C05385=1038.334,449.615,-148.521,176.484,47.158,159.856
C05386=1038.308,449.370,-148.478,176.465,47.152,159.852
C05387=1038.284,449.126,-148.433,176.446,47.146,159.848
C05388=1038.259,448.881,-148.389,176.428,47.139,159.843
C05389=1038.236,448.635,-148.344,176.409,47.132,159.839
C05390=1038.213,448.391,-148.298,176.390,47.125,159.834
C05391=1038.190,448.146,-148.252,176.372,47.118,159.830
C05392=1038.168,447.901,-148.206,176.353,47.112,159.825
C05393=1038.146,447.657,-148.159,176.335,47.105,159.821
C05394=1038.125,447.413,-148.112,176.318,47.097,159.816
C05395=1038.105,447.168,-148.064,176.299,47.090,159.812
C05396=1038.085,446.924,-148.016,176.281,47.083,159.807
C05397=1038.065,446.680,-147.967,176.264,47.076,159.803
C05398=1038.047,446.435,-147.918,176.245,47.068,159.798
C05399=1038.029,446.191,-147.869,176.228,47.060,159.794
C05400=1038.012,445.948,-147.819,176.211,47.053,159.789
C05401=1037.994,445.705,-147.768,176.192,47.045,159.785
C05402=1037.978,445.460,-147.718,176.174,47.037,159.780
C05403=1037.962,445.217,-147.666,176.157,47.029,159.776
C05404=1037.946,444.973,-147.614,176.141,47.021,159.771
C05405=1037.932,444.730,-147.563,176.123,47.013,159.766
C05406=1037.917,444.485,-147.509,176.105,47.005,159.762
C05407=1037.904,444.241,-147.456,176.089,46.996,159.757
C05408=1037.890,443.996,-147.402,176.071,46.988,159.752
C05409=1037.877,443.752,-147.349,176.054,46.979,159.747
C05410=1037.863,443.508,-147.296,176.038,46.971,159.743
C05411=1037.849,443.264,-147.243,176.020,46.963,159.738
C05412=1037.836,443.020,-147.189,176.004,46.955,159.734
C05413=1037.823,442.776,-147.136,175.987,46.946,159.729
C05414=1037.810,442.532,-147.082,175.971,46.938,159.725
C05415=1037.797,442.288,-147.029,175.954,46.930,159.720
C05416=1037.783,442.044,-146.977,175.937,46.922,159.716
C05417=1037.770,441.800,-146.924,175.920,46.914,159.711
C05418=1037.757,441.556,-146.871,175.904,46.905,159.707
C05419=1037.744,441.312,-146.818,175.888,46.897,159.702
C05420=1037.732,441.068,-146.766,175.871,46.889,159.698
C05421=1037.718,440.824,-146.712,175.855,46.881,159.693
C05422=1037.705,440.581,-146.660,175.839,46.873,159.689
C05423=1037.692,440.336,-146.607,175.824,46.865,159.685
C05424=1037.679,440.091,-146.555,175.807,46.857,159.680
C05425=1037.667,439.848,-146.502,175.791,46.849,159.676
C05426=1037.653,439.604,-146.450,175.775,46.841,159.671
C05427=1037.640,439.359,-146.398,175.759,46.833,159.667
C05428=1037.628,439.115,-146.346,175.744,46.825,159.663
C05429=1037.615,438.871,-146.293,175.728,46.817,159.659
C05430=1037.602,438.627,-146.241,175.712,46.809,159.654
C05431=1037.590,438.383,-146.189,175.697,46.802,159.650
C05432=1037.577,438.138,-146.137,175.681,46.794,159.646
C05433=1037.564,437.895,-146.085,175.665,46.786,159.642
C05434=1037.552,437.653,-146.034,175.650,46.778,159.638
C05435=1037.539,437.412,-145.983,175.635,46.771,159.634
C05436=1037.527,437.170,-145.931,175.619,46.763,159.629
C05437=1037.514,436.929,-145.880,175.605,46.755,159.625
C05438=1037.502,436.688,-145.829,175.590,46.748,159.621
C05439=1037.489,436.446,-145.778,175.574,46.740,159.617
C05440=1037.477,436.205,-145.726,175.560,46.733,159.613
C05441=1037.465,435.963,-145.676,175.545,46.725,159.609
C05442=1037.453,435.719,-145.624,175.530,46.718,159.605
C05443=1037.439,435.474,-145.573,175.514,46.710,159.601
C05444=1037.428,435.230,-145.521,175.500,46.703,159.597
C05445=1037.416,434.985,-145.470,175.485,46.696,159.593
C05446=1037.403,434.741,-145.419,175.470,46.688,159.589
C05447=1037.391,434.497,-145.368,175.455,46.681,159.585
C05448=1037.379,434.252,-145.317,175.440,46.673,159.581
C05449=1037.365,434.007,-145.266,175.426,46.666,159.577
C05450=1037.353,433.763,-145.214,175.411,46.658,159.574
C05451=1037.341,433.519,-145.164,175.397,46.651,159.570
C05452=1037.329,433.274,-145.113,175.382,46.644,159.566
C05453=1037.317,433.029,-145.062,175.368,46.637,159.562
C05454=1037.304,432.785,-145.011,175.354,46.629,159.558
C05455=1037.292,432.540,-144.961,175.339,46.622,159.554
C05456=1037.280,432.297,-144.910,175.325,46.615,159.551
C05457=1037.268,432.052,-144.860,175.310,46.607,159.547
C05458=1037.256,431.807,-144.809,175.296,46.601,159.543
C05459=1037.244,431.562,-144.758,175.283,46.593,159.539
C05460=1037.232,431.317,-144.708,175.268,46.586,159.535
C05461=1037.220,431.072,-144.658,175.254,46.579,159.532
C05462=1037.208,430.829,-144.607,175.240,46.572,159.528
C05463=1037.196,430.584,-144.557,175.226,46.565,159.524
C05464=1037.184,430.339,-144.506,175.213,46.558,159.521
C05465=1037.173,430.095,-144.456,175.199,46.551,159.517
C05466=1037.161,429.850,-144.406,175.184,46.544,159.513
C05467=1037.149,429.606,-144.356,175.171,46.537,159.510
C05468=1037.138,429.360,-144.306,175.157,46.530,159.506
C05469=1037.125,429.116,-144.256,175.144,46.523,159.502
C05470=1037.114,428.871,-144.207,175.130,46.516,159.499
C05471=1037.103,428.626,-144.156,175.117,46.509,159.495
C05472=1037.091,428.382,-144.106,175.103,46.503,159.492
C05473=1037.080,428.137,-144.056,175.090,46.495,159.488
C05474=1037.068,427.892,-144.006,175.076,46.489,159.485
C05475=1037.056,427.648,-143.957,175.063,46.482,159.481
C05476=1037.044,427.402,-143.907,175.049,46.475,159.478
C05477=1037.033,427.157,-143.858,175.036,46.468,159.474
C05478=1037.022,426.913,-143.808,175.023,46.462,159.471
C05479=1037.010,426.668,-143.759,175.010,46.455,159.467
C05480=1036.998,426.423,-143.710,174.997,46.448,159.464
C05481=1036.987,426.178,-143.661,174.984,46.442,159.460
C05482=1036.975,425.933,-143.611,174.970,46.435,159.457
C05483=1036.963,425.689,-143.561,174.957,46.428,159.453
C05484=1036.952,425.444,-143.512,174.944,46.422,159.450
C05485=1036.941,425.199,-143.463,174.932,46.415,159.447
C05486=1036.930,424.953,-143.415,174.919,46.409,159.443
C05487=1036.918,424.709,-143.366,174.905,46.402,159.440
C05488=1036.907,424.464,-143.316,174.892,46.395,159.436
C05489=1036.896,424.219,-143.267,174.880,46.389,159.433
C05490=1036.884,423.974,-143.218,174.867,46.383,159.430
C05491=1036.873,423.730,-143.169,174.855,46.376,159.427
C05492=1036.861,423.484,-143.121,174.842,46.370,159.423
C05493=1036.850,423.239,-143.072,174.830,46.364,159.420
C05494=1036.839,423.000,-143.024,174.817,46.357,159.417
C05495=1036.828,422.760,-142.977,174.805,46.351,159.414
C05496=1036.817,422.521,-142.930,174.793,46.345,159.411
C05497=1036.806,422.281,-142.882,174.781,46.339,159.408
C05498=1036.795,422.041,-142.835,174.769,46.333,159.404
C05499=1036.784,421.802,-142.788,174.756,46.326,159.401
C05500=1036.774,421.562,-142.741,174.745,46.320,159.398
C05501=1036.763,421.322,-142.693,174.732,46.314,159.395
C05502=1036.752,421.077,-142.645,174.720,46.308,159.392
C05503=1036.740,420.833,-142.598,174.708,46.302,159.389
C05504=1036.729,420.588,-142.549,174.696,46.296,159.386
C05505=1036.718,420.343,-142.500,174.684,46.290,159.382
C05506=1036.708,420.097,-142.453,174.672,46.283,159.379
C05507=1036.697,419.852,-142.405,174.659,46.278,159.376
C05508=1036.685,419.607,-142.356,174.648,46.271,159.373
C05509=1036.675,419.362,-142.309,174.636,46.265,159.370
C05510=1036.664,419.117,-142.260,174.623,46.259,159.367
C05511=1036.653,418.871,-142.212,174.612,46.253,159.364
C05512=1036.642,418.626,-142.165,174.600,46.247,159.361
C05513=1036.631,418.381,-142.117,174.589,46.241,159.358
C05514=1036.620,418.136,-142.069,174.576,46.235,159.355
C05515=1036.610,417.891,-142.022,174.565,46.229,159.352
C05516=1036.599,417.646,-141.974,174.553,46.223,159.349
C05517=1036.589,417.400,-141.926,174.541,46.217,159.346
C05518=1036.577,417.155,-141.879,174.530,46.211,159.343
C05519=1036.567,416.910,-141.831,174.518,46.205,159.340
C05520=1036.556,416.664,-141.784,174.507,46.200,159.337
C05521=1036.545,416.419,-141.737,174.496,46.194,159.334
C05522=1036.535,416.174,-141.689,174.484,46.188,159.331
C05523=1036.523,415.929,-141.642,174.473,46.182,159.328
C05524=1036.513,415.683,-141.595,174.461,46.177,159.325
C05525=1036.503,415.438,-141.548,174.450,46.171,159.322
C05526=1036.491,415.192,-141.501,174.439,46.165,159.320
C05527=1036.481,414.947,-141.454,174.427,46.160,159.317
C05528=1036.470,414.702,-141.407,174.416,46.154,159.314
C05529=1036.460,414.457,-141.360,174.405,46.148,159.311
C05530=1036.450,414.212,-141.313,174.393,46.142,159.308
C05531=1036.438,413.965,-141.266,174.382,46.137,159.305
C05532=1036.428,413.720,-141.219,174.371,46.131,159.303
C05533=1036.417,413.475,-141.173,174.360,46.126,159.300
C05534=1036.407,413.230,-141.125,174.349,46.120,159.297
C05535=1036.397,412.984,-141.079,174.337,46.114,159.294
C05536=1036.386,412.739,-141.032,174.327,46.109,159.291
C05537=1036.376,412.494,-140.985,174.316,46.103,159.289
C05538=1036.365,412.248,-140.939,174.305,46.098,159.286
C05539=1036.355,412.003,-140.892,174.294,46.093,159.283
C05540=1036.345,411.757,-140.845,174.284,46.087,159.281
C05541=1036.334,411.512,-140.799,174.272,46.082,159.278
C05542=1036.325,411.266,-140.752,174.261,46.076,159.275
C05543=1036.314,411.020,-140.706,174.250,46.070,159.272
C05544=1036.303,410.775,-140.660,174.240,46.065,159.270
C05545=1036.293,410.529,-140.614,174.229,46.060,159.267
C05546=1036.283,410.285,-140.568,174.218,46.055,159.264
C05547=1036.272,410.039,-140.522,174.208,46.049,159.262
C05548=1036.262,409.793,-140.476,174.197,46.044,159.259
C05549=1036.252,409.547,-140.429,174.186,46.039,159.256
C05550=1036.241,409.302,-140.383,174.176,46.034,159.254
C05551=1036.231,409.057,-140.338,174.165,46.028,159.251
C05552=1036.221,408.811,-140.293,174.155,46.023,159.249
C05553=1036.211,408.565,-140.246,174.145,46.018,159.246
C05554=1036.201,408.330,-140.202,174.135,46.013,159.244
C05555=1036.192,408.095,-140.159,174.124,46.008,159.241
C05556=1036.181,407.860,-140.114,174.115,46.003,159.239
C05557=1036.172,407.624,-140.071,174.105,45.998,159.236
C05558=1036.162,407.390,-140.028,174.095,45.993,159.234
C05559=1036.152,407.155,-139.984,174.085,45.988,159.231
C05560=1036.144,406.919,-139.940,174.076,45.983,159.229
C05561=1036.133,406.683,-139.896,174.065,45.979,159.227
C05562=1036.123,406.439,-139.850,174.056,45.973,159.224
C05563=1036.113,406.192,-139.805,174.045,45.968,159.222
C05564=1036.103,405.947,-139.760,174.035,45.963,159.219
C05565=1036.093,405.701,-139.714,174.025,45.959,159.217
C05566=1036.084,405.455,-139.669,174.015,45.953,159.214
C05567=1036.074,405.211,-139.623,174.005,45.948,159.212
C05568=1036.063,404.964,-139.578,173.995,45.944,159.209
C05569=1036.054,404.719,-139.533,173.985,45.938,159.207
C05570=1036.044,404.474,-139.487,173.975,45.933,159.204
C05571=1036.034,404.227,-139.442,173.964,45.929,159.202
C05572=1036.024,403.982,-139.397,173.955,45.923,159.199
C05573=1036.015,403.736,-139.352,173.945,45.919,159.197
C05574=1036.005,403.490,-139.307,173.936,45.914,159.195
C05575=1035.995,403.244,-139.262,173.925,45.909,159.192
C05576=1035.986,402.999,-139.217,173.916,45.904,159.190
C05577=1035.976,402.753,-139.172,173.906,45.899,159.188
C05578=1035.966,402.508,-139.127,173.896,45.894,159.185
C05579=1035.956,402.262,-139.082,173.886,45.889,159.183
C05580=1035.946,402.016,-139.037,173.877,45.885,159.181
C05581=1035.936,401.771,-138.993,173.867,45.880,159.178
C05582=1035.927,401.525,-138.948,173.858,45.875,159.176
C05583=1035.917,401.279,-138.904,173.848,45.871,159.174
C05584=1035.908,401.033,-138.859,173.838,45.866,159.171
C05585=1035.898,400.788,-138.814,173.828,45.861,159.169
C05586=1035.889,400.542,-138.770,173.819,45.856,159.167
C05587=1035.879,400.296,-138.725,173.809,45.852,159.164
C05588=1035.869,400.050,-138.681,173.800,45.848,159.162
C05589=1035.860,399.805,-138.636,173.791,45.843,159.160
C05590=1035.850,399.558,-138.592,173.781,45.838,159.158
C05591=1035.841,399.313,-138.547,173.772,45.833,159.155
C05592=1035.830,399.067,-138.504,173.763,45.829,159.153
C05593=1035.821,398.822,-138.459,173.753,45.825,159.151
C05594=1035.811,398.575,-138.415,173.743,45.820,159.149
C05595=1035.802,398.329,-138.371,173.735,45.815,159.146
C05596=1035.792,398.083,-138.327,173.724,45.811,159.144
C05597=1035.783,397.838,-138.283,173.716,45.807,159.142
C05598=1035.773,397.593,-138.239,173.707,45.802,159.140
C05599=1035.764,397.346,-138.194,173.697,45.798,159.138
C05600=1035.754,397.100,-138.150,173.688,45.793,159.135
C05601=1035.744,396.854,-138.107,173.679,45.789,159.133
C05602=1035.735,396.609,-138.063,173.670,45.784,159.131
C05603=1035.726,396.363,-138.019,173.661,45.780,159.129
C05604=1035.717,396.117,-137.975,173.651,45.776,159.127
C05605=1035.706,395.871,-137.931,173.642,45.772,159.125
C05606=1035.698,395.626,-137.888,173.633,45.767,159.122
C05607=1035.688,395.379,-137.843,173.624,45.762,159.120
C05608=1035.679,395.133,-137.800,173.615,45.758,159.118
C05609=1035.670,394.888,-137.757,173.606,45.754,159.116
C05610=1035.660,394.641,-137.713,173.597,45.750,159.114
C05611=1035.651,394.396,-137.669,173.588,45.745,159.112
C05612=1035.642,394.150,-137.626,173.579,45.741,159.110
C05613=1035.632,393.903,-137.582,173.570,45.737,159.108
C05614=1035.623,393.678,-137.543,173.563,45.733,159.106
C05615=1035.616,393.453,-137.503,173.554,45.729,159.104
C05616=1035.607,393.228,-137.464,173.545,45.725,159.102
C05617=1035.598,393.003,-137.424,173.538,45.722,159.100
C05618=1035.590,392.778,-137.384,173.530,45.718,159.098
C05619=1035.581,392.553,-137.345,173.522,45.714,159.097
C05620=1035.573,392.328,-137.305,173.514,45.710,159.095
C05621=1035.565,392.103,-137.265,173.506,45.706,159.093
C05622=1035.555,391.857,-137.223,173.497,45.702,159.091
C05623=1035.546,391.611,-137.179,173.489,45.698,159.089
C05624=1035.537,391.366,-137.136,173.480,45.694,159.087
C05625=1035.528,391.120,-137.093,173.471,45.690,159.085
C05626=1035.519,390.873,-137.050,173.462,45.686,159.083
C05627=1035.510,390.627,-137.007,173.454,45.682,159.081
C05628=1035.501,390.380,-136.964,173.445,45.678,159.079
C05629=1035.491,390.135,-136.922,173.436,45.674,159.077
C05630=1035.482,389.889,-136.879,173.428,45.670,159.075
C05631=1035.473,389.642,-136.836,173.419,45.667,159.073
C05632=1035.464,389.396,-136.793,173.412,45.662,159.071
C05633=1035.455,389.150,-136.750,173.403,45.658,159.069
C05634=1035.446,388.905,-136.708,173.394,45.654,159.067
C05635=1035.436,388.658,-136.665,173.386,45.651,159.065
C05636=1035.428,388.412,-136.622,173.377,45.647,159.063
C05637=1035.419,388.166,-136.580,173.369,45.642,159.061
C05638=1035.410,387.920,-136.537,173.361,45.638,159.060
C05639=1035.401,387.674,-136.495,173.353,45.635,159.058
C05640=1035.391,387.427,-136.452,173.344,45.631,159.056
C05641=1035.383,387.181,-136.409,173.335,45.627,159.054
C05642=1035.374,386.935,-136.367,173.327,45.623,159.052
C05643=1035.365,386.689,-136.325,173.320,45.620,159.050
C05644=1035.356,386.443,-136.283,173.311,45.616,159.048
C05645=1035.346,386.197,-136.241,173.303,45.612,159.046
C05646=1035.337,385.950,-136.199,173.294,45.608,159.045
C05647=1035.328,385.704,-136.156,173.287,45.605,159.043
C05648=1035.319,385.458,-136.114,173.278,45.601,159.041
C05649=1035.311,385.211,-136.072,173.270,45.597,159.039
C05650=1035.301,384.966,-136.030,173.261,45.594,159.037
C05651=1035.292,384.719,-135.988,173.254,45.590,159.036
C05652=1035.283,384.473,-135.946,173.245,45.586,159.034
C05653=1035.274,384.226,-135.905,173.237,45.583,159.032
C05654=1035.265,383.981,-135.862,173.230,45.579,159.030
C05655=1035.256,383.734,-135.820,173.221,45.576,159.028
C05656=1035.248,383.488,-135.778,173.213,45.572,159.027
C05657=1035.239,383.241,-135.736,173.206,45.568,159.025
C05658=1035.230,382.995,-135.695,173.197,45.565,159.023
C05659=1035.222,382.749,-135.653,173.190,45.561,159.021
C05660=1035.213,382.503,-135.612,173.181,45.557,159.019
C05661=1035.204,382.257,-135.570,173.173,45.554,159.018
C05662=1035.195,382.010,-135.528,173.166,45.551,159.016
C05663=1035.186,381.764,-135.486,173.157,45.547,159.014
C05664=1035.177,381.517,-135.445,173.150,45.543,159.012
C05665=1035.170,381.271,-135.403,173.142,45.540,159.011
C05666=1035.161,381.025,-135.361,173.135,45.537,159.009
C05667=1035.152,380.779,-135.319,173.126,45.533,159.007
C05668=1035.143,380.532,-135.278,173.119,45.529,159.006
C05669=1035.135,380.286,-135.237,173.111,45.526,159.004
C05670=1035.126,380.040,-135.195,173.104,45.523,159.002
C05671=1035.117,379.793,-135.154,173.095,45.519,159.001
C05672=1035.108,379.547,-135.112,173.088,45.516,158.999
C05673=1035.100,379.301,-135.071,173.080,45.512,158.997
C05674=1035.085,378.885,-135.001,173.067,45.506,158.994
C05675=1035.071,378.470,-134.931,173.054,45.501,158.992
C05676=1035.057,378.055,-134.862,173.042,45.495,158.989
C05677=1035.043,377.640,-134.792,173.029,45.490,158.986
C05678=1035.033,377.393,-134.752,173.021,45.487,158.984
C05679=1035.025,377.147,-134.711,173.014,45.483,158.983
C05680=1035.017,376.900,-134.670,173.005,45.480,158.981
C05681=1035.008,376.653,-134.628,172.998,45.477,158.980
C05682=1035.000,376.407,-134.588,172.991,45.473,158.978
C05683=1034.990,376.160,-134.547,172.983,45.470,158.976
C05684=1034.982,375.914,-134.507,172.976,45.467,158.975
C05685=1034.974,375.667,-134.466,172.968,45.464,158.973
C05686=1034.965,375.421,-134.424,172.961,45.461,158.972
C05687=1034.956,375.175,-134.384,172.954,45.457,158.970
C05688=1034.948,374.929,-134.343,172.946,45.455,158.968
C05689=1034.939,374.682,-134.302,172.939,45.451,158.967
C05690=1034.931,374.435,-134.262,172.932,45.448,158.965
C05691=1034.922,374.189,-134.222,172.924,45.445,158.964
C05692=1034.914,373.942,-134.181,172.916,45.442,158.962
C05693=1034.906,373.696,-134.140,172.909,45.439,158.961
C05694=1034.897,373.449,-134.099,172.902,45.436,158.959
C05695=1034.889,373.202,-134.060,172.895,45.433,158.957
C05696=1034.881,372.956,-134.019,172.887,45.430,158.956
C05697=1034.872,372.709,-133.978,172.880,45.426,158.954
C05698=1034.863,372.463,-133.938,172.873,45.423,158.953
C05699=1034.855,372.217,-133.897,172.866,45.421,158.951
C05700=1034.847,371.969,-133.857,172.858,45.418,158.950
C05701=1034.839,371.723,-133.816,172.851,45.414,158.948
C05702=1034.830,371.477,-133.776,172.844,45.411,158.947
C05703=1034.822,371.231,-133.736,172.837,45.408,158.945
C05704=1034.814,370.983,-133.696,172.830,45.405,158.944
C05705=1034.806,370.737,-133.655,172.823,45.402,158.942
C05706=1034.797,370.490,-133.616,172.815,45.400,158.941
C05707=1034.789,370.244,-133.575,172.809,45.397,158.939
C05708=1034.781,369.998,-133.534,172.802,45.394,158.938
C05709=1034.773,369.751,-133.495,172.795,45.391,158.936
C05710=1034.764,369.503,-133.455,172.788,45.388,158.935
C05711=1034.756,369.257,-133.415,172.781,45.385,158.933
C05712=1034.748,369.011,-133.375,172.774,45.382,158.932
C05713=1034.740,368.764,-133.335,172.766,45.379,158.930
C05714=1034.731,368.518,-133.295,172.759,45.377,158.929
C05715=1034.723,368.271,-133.255,172.752,45.374,158.928
C05716=1034.714,368.024,-133.216,172.745,45.371,158.926
C05717=1034.706,367.777,-133.176,172.739,45.368,158.925
C05718=1034.698,367.531,-133.136,172.732,45.366,158.924
C05719=1034.689,367.284,-133.096,172.725,45.363,158.922
C05720=1034.681,367.037,-133.057,172.718,45.360,158.921
C05721=1034.673,366.791,-133.017,172.711,45.357,158.919
C05722=1034.665,366.544,-132.977,172.704,45.354,158.918
C05723=1034.657,366.297,-132.938,172.698,45.351,158.916
C05724=1034.648,366.051,-132.899,172.691,45.349,158.915
C05725=1034.641,365.804,-132.859,172.684,45.346,158.914
C05726=1034.632,365.557,-132.819,172.677,45.343,158.912
C05727=1034.624,365.310,-132.780,172.670,45.340,158.911
C05728=1034.616,365.064,-132.740,172.664,45.338,158.910
C05729=1034.607,364.817,-132.701,172.657,45.335,158.908
C05730=1034.595,364.422,-132.638,172.646,45.331,158.906
C05731=1034.582,364.028,-132.575,172.635,45.327,158.904
C05732=1034.569,363.633,-132.512,172.624,45.322,158.902
C05733=1034.557,363.238,-132.449,172.614,45.318,158.899
C05734=1034.548,362.991,-132.409,172.607,45.316,158.898
C05735=1034.540,362.745,-132.370,172.600,45.313,158.897
C05736=1034.533,362.498,-132.331,172.593,45.310,158.895
C05737=1034.524,362.251,-132.292,172.587,45.308,158.894
C05738=1034.516,362.005,-132.253,172.580,45.306,158.893
C05739=1034.509,361.757,-132.213,172.573,45.303,158.892
C05740=1034.501,361.511,-132.174,172.567,45.300,158.890
C05741=1034.492,361.264,-132.136,172.561,45.297,158.889
C05742=1034.484,361.017,-132.097,172.554,45.295,158.888
C05743=1034.477,360.770,-132.057,172.548,45.293,158.886
C05744=1034.468,360.523,-132.018,172.541,45.290,158.885
C05745=1034.461,360.277,-131.980,172.534,45.288,158.884
C05746=1034.452,360.030,-131.941,172.528,45.285,158.882
C05747=1034.444,359.783,-131.902,172.521,45.283,158.881
C05748=1034.436,359.536,-131.864,172.515,45.280,158.880
C05749=1034.428,359.289,-131.825,172.509,45.278,158.879
C05750=1034.420,359.042,-131.786,172.502,45.276,158.877
C05751=1034.412,358.795,-131.747,172.495,45.273,158.876
C05752=1034.404,358.549,-131.709,172.489,45.271,158.875
C05753=1034.396,358.302,-131.670,172.482,45.269,158.874
C05754=1034.388,358.055,-131.632,172.477,45.266,158.873
C05755=1034.380,357.808,-131.593,172.470,45.264,158.871
C05756=1034.372,357.561,-131.555,172.463,45.261,158.870
C05757=1034.365,357.314,-131.516,172.457,45.259,158.869
C05758=1034.357,357.067,-131.477,172.451,45.257,158.868
C05759=1034.349,356.821,-131.438,172.445,45.254,158.866
C05760=1034.341,356.574,-131.400,172.438,45.252,158.865
C05761=1034.333,356.326,-131.361,172.432,45.250,158.864
C05762=1034.325,356.080,-131.323,172.426,45.248,158.863
C05763=1034.318,355.832,-131.285,172.420,45.245,158.861
C05764=1034.310,355.586,-131.247,172.413,45.243,158.860
C05765=1034.301,355.339,-131.209,172.407,45.241,158.859
C05766=1034.294,355.092,-131.170,172.401,45.238,158.858
C05767=1034.285,354.845,-131.132,172.395,45.236,158.857
C05768=1034.278,354.598,-131.094,172.388,45.234,158.855
C05769=1034.270,354.351,-131.056,172.382,45.232,158.854
C05770=1034.263,354.104,-131.017,172.376,45.229,158.853
C05771=1034.254,353.857,-130.979,172.370,45.228,158.852
C05772=1034.246,353.610,-130.942,172.363,45.225,158.851
C05773=1034.239,353.363,-130.904,172.358,45.223,158.850
C05774=1034.231,353.116,-130.865,172.351,45.221,158.848
C05775=1034.223,352.869,-130.828,172.345,45.219,158.847
C05776=1034.215,352.622,-130.789,172.339,45.217,158.846
C05777=1034.207,352.375,-130.752,172.333,45.214,158.845
C05778=1034.200,352.129,-130.714,172.326,45.212,158.844
C05779=1034.192,351.881,-130.676,172.321,45.210,158.843
C05780=1034.184,351.634,-130.638,172.314,45.208,158.842
C05781=1034.177,351.387,-130.600,172.308,45.206,158.840
C05782=1034.169,351.140,-130.562,172.303,45.204,158.839
C05783=1034.161,350.893,-130.525,172.296,45.202,158.838
C05784=1034.153,350.647,-130.486,172.291,45.199,158.837
C05785=1034.146,350.399,-130.448,172.284,45.198,158.836
C05786=1034.134,350.011,-130.389,172.275,45.194,158.834
C05787=1034.121,349.622,-130.330,172.266,45.191,158.833
C05788=1034.110,349.233,-130.271,172.256,45.188,158.831
C05789=1034.097,348.844,-130.212,172.246,45.185,158.829
C05790=1034.090,348.597,-130.174,172.241,45.183,158.828
C05791=1034.082,348.351,-130.136,172.235,45.181,158.827
C05792=1034.075,348.104,-130.099,172.229,45.179,158.826
C05793=1034.067,347.857,-130.062,172.223,45.177,158.825
C05794=1034.059,347.609,-130.024,172.217,45.175,158.824
C05795=1034.051,347.362,-129.987,172.211,45.173,158.823
C05796=1034.044,347.115,-129.950,172.205,45.171,158.822
C05797=1034.036,346.868,-129.913,172.200,45.169,158.820
C05798=1034.028,346.621,-129.875,172.193,45.167,158.819
C05799=1034.021,346.374,-129.838,172.188,45.165,158.818
C05800=1034.013,346.127,-129.801,172.182,45.163,158.817
C05801=1034.005,345.880,-129.763,172.176,45.161,158.816
C05802=1033.997,345.633,-129.726,172.170,45.160,158.815
C05803=1033.990,345.386,-129.688,172.165,45.158,158.814
C05804=1033.982,345.138,-129.652,172.158,45.156,158.813
C05805=1033.975,344.891,-129.615,172.153,45.154,158.812
C05806=1033.967,344.644,-129.578,172.147,45.152,158.811
C05807=1033.960,344.397,-129.540,172.142,45.151,158.810
C05808=1033.952,344.150,-129.503,172.136,45.149,158.809
C05809=1033.945,343.902,-129.466,172.130,45.147,158.808
C05810=1033.936,343.603,-129.422,172.124,45.145,158.807
C05811=1033.926,343.303,-129.376,172.116,45.143,158.806
C05812=1033.917,343.003,-129.331,172.109,45.140,158.804
C05813=1033.908,342.703,-129.287,172.103,45.138,158.803
C05814=1033.901,342.456,-129.250,172.097,45.136,158.802
C05815=1033.893,342.209,-129.214,172.091,45.134,158.801
C05816=1033.886,341.962,-129.176,172.085,45.133,158.800
C05817=1033.878,341.715,-129.139,172.080,45.131,158.799
C05818=1033.871,341.467,-129.103,172.075,45.129,158.798
C05819=1033.863,341.220,-129.065,172.068,45.127,158.797
C05820=1033.856,340.973,-129.029,172.063,45.126,158.796
C05821=1033.849,340.725,-128.992,172.057,45.124,158.795
C05822=1033.841,340.478,-128.955,172.052,45.123,158.794
C05823=1033.833,340.231,-128.919,172.046,45.120,158.793
C05824=1033.825,339.984,-128.882,172.040,45.119,158.792
C05825=1033.818,339.737,-128.846,172.035,45.118,158.791
C05826=1033.811,339.490,-128.810,172.029,45.116,158.790
C05827=1033.803,339.242,-128.773,172.024,45.114,158.789
C05828=1033.795,338.995,-128.736,172.019,45.113,158.789
C05829=1033.788,338.748,-128.700,172.012,45.111,158.787
C05830=1033.780,338.500,-128.664,172.007,45.109,158.787
C05831=1033.774,338.253,-128.628,172.002,45.108,158.786
C05832=1033.766,338.007,-128.591,171.996,45.107,158.785
C05833=1033.758,337.759,-128.554,171.991,45.104,158.784
C05834=1033.750,337.512,-128.518,171.986,45.103,158.783
C05835=1033.743,337.265,-128.482,171.980,45.102,158.782
C05836=1033.736,337.017,-128.446,171.975,45.100,158.781
C05837=1033.729,336.770,-128.409,171.969,45.098,158.780
C05838=1033.721,336.522,-128.373,171.964,45.096,158.779
C05839=1033.714,336.275,-128.337,171.958,45.095,158.778
C05840=1033.706,336.028,-128.301,171.953,45.094,158.777
C05841=1033.699,335.781,-128.265,171.948,45.092,158.776
C05842=1033.689,335.442,-128.215,171.940,45.090,158.775
C05843=1033.679,335.103,-128.165,171.933,45.088,158.774
C05844=1033.669,334.764,-128.116,171.925,45.086,158.773
C05845=1033.659,334.424,-128.066,171.918,45.084,158.771
C05846=1033.651,334.177,-128.030,171.913,45.082,158.770
C05847=1033.644,333.930,-127.994,171.907,45.081,158.770
C05848=1033.636,333.682,-127.958,171.902,45.079,158.769
C05849=1033.629,333.434,-127.923,171.896,45.078,158.768
C05850=1033.622,333.188,-127.887,171.892,45.077,158.767
C05851=1033.614,332.941,-127.851,171.886,45.075,158.766
C05852=1033.606,332.694,-127.815,171.881,45.074,158.765
C05853=1033.599,332.446,-127.780,171.875,45.073,158.764
C05854=1033.592,332.199,-127.744,171.870,45.071,158.764
C05855=1033.584,331.952,-127.708,171.865,45.069,158.763
C05856=1033.577,331.703,-127.672,171.860,45.068,158.762
C05857=1033.570,331.457,-127.636,171.854,45.067,158.761
C05858=1033.563,331.209,-127.601,171.849,45.066,158.760
C05859=1033.555,330.962,-127.565,171.844,45.064,158.759
C05860=1033.548,330.714,-127.530,171.839,45.063,158.758
C05861=1033.541,330.467,-127.494,171.834,45.061,158.758
C05862=1033.533,330.220,-127.457,171.829,45.060,158.757
C05863=1033.526,329.973,-127.423,171.823,45.059,158.756
C05864=1033.518,329.725,-127.387,171.818,45.057,158.755
C05865=1033.511,329.478,-127.352,171.813,45.056,158.754
C05866=1033.505,329.230,-127.316,171.808,45.055,158.754
C05867=1033.497,328.983,-127.280,171.803,45.053,158.753
C05868=1033.490,328.736,-127.245,171.798,45.052,158.752
C05869=1033.483,328.488,-127.209,171.792,45.051,158.751
C05870=1033.476,328.241,-127.174,171.787,45.050,158.750
C05871=1033.468,327.993,-127.139,171.782,45.048,158.749
C05872=1033.461,327.746,-127.104,171.777,45.047,158.749
C05873=1033.453,327.499,-127.068,171.772,45.046,158.748
C05874=1033.446,327.251,-127.033,171.767,45.045,158.747
C05875=1033.438,327.004,-126.998,171.761,45.043,158.746
C05876=1033.431,326.756,-126.963,171.756,45.043,158.745
C05877=1033.423,326.509,-126.928,171.751,45.041,158.745
C05878=1033.416,326.261,-126.893,171.746,45.040,158.744
C05879=1033.408,326.014,-126.858,171.742,45.039,158.743
C05880=1033.402,325.767,-126.823,171.737,45.038,158.742
C05881=1033.394,325.519,-126.788,171.732,45.037,158.742
C05882=1033.387,325.271,-126.753,171.727,45.035,158.741
C05883=1033.379,325.024,-126.719,171.721,45.034,158.740
C05884=1033.372,324.776,-126.683,171.716,45.034,158.739
C05885=1033.364,324.529,-126.649,171.711,45.032,158.738
C05886=1033.358,324.282,-126.613,171.706,45.031,158.738
C05887=1033.350,324.034,-126.579,171.701,45.030,158.737
C05888=1033.343,323.787,-126.543,171.696,45.029,158.736
C05889=1033.335,323.540,-126.509,171.691,45.028,158.735
C05890=1033.328,323.293,-126.474,171.687,45.027,158.735
C05891=1033.320,323.045,-126.439,171.682,45.026,158.734
C05892=1033.313,322.798,-126.404,171.677,45.024,158.733
C05893=1033.306,322.550,-126.370,171.672,45.023,158.732
C05894=1033.299,322.303,-126.335,171.666,45.023,158.732
C05895=1033.292,322.054,-126.300,171.661,45.022,158.731
C05896=1033.284,321.807,-126.265,171.656,45.020,158.730
C05897=1033.277,321.560,-126.230,171.651,45.019,158.729
C05898=1033.266,321.164,-126.176,171.644,45.017,158.728
C05899=1033.254,320.767,-126.119,171.636,45.016,158.727
C05900=1033.243,320.371,-126.064,171.628,45.014,158.726
C05901=1033.231,319.974,-126.009,171.621,45.013,158.725
C05902=1033.224,319.726,-125.974,171.616,45.012,158.724
C05903=1033.217,319.479,-125.939,171.611,45.011,158.723
C05904=1033.210,319.231,-125.905,171.607,45.010,158.723
C05905=1033.203,318.984,-125.870,171.601,45.008,158.722
C05906=1033.196,318.736,-125.836,171.597,45.007,158.721
C05907=1033.189,318.489,-125.801,171.592,45.006,158.720
C05908=1033.181,318.242,-125.767,171.587,45.005,158.720
C05909=1033.175,317.994,-125.733,171.582,45.004,158.719
C05910=1033.167,317.747,-125.698,171.577,45.004,158.718
C05911=1033.161,317.499,-125.664,171.573,45.003,158.718
C05912=1033.153,317.252,-125.629,171.568,45.002,158.717
C05913=1033.146,317.004,-125.595,171.563,45.001,158.716
C05914=1033.139,316.756,-125.561,171.558,45.000,158.716
C05915=1033.132,316.509,-125.526,171.553,44.999,158.715
C05916=1033.125,316.261,-125.492,171.549,44.998,158.714
C05917=1033.118,316.014,-125.457,171.544,44.997,158.713
C05918=1033.112,315.766,-125.423,171.539,44.996,158.713
C05919=1033.104,315.519,-125.389,171.534,44.995,158.712
C05920=1033.097,315.272,-125.355,171.529,44.994,158.711
C05921=1033.090,315.024,-125.320,171.525,44.993,158.711
C05922=1033.083,314.776,-125.286,171.521,44.992,158.710
C05923=1033.077,314.529,-125.251,171.516,44.992,158.709
C05924=1033.070,314.282,-125.218,171.511,44.991,158.709
C05925=1033.063,314.034,-125.184,171.506,44.990,158.708
C05926=1033.056,313.787,-125.149,171.502,44.989,158.707
C05927=1033.049,313.539,-125.115,171.497,44.988,158.707
C05928=1033.041,313.291,-125.081,171.492,44.987,158.706
C05929=1033.036,313.044,-125.047,171.488,44.986,158.705
C05930=1033.028,312.796,-125.013,171.484,44.985,158.705
C05931=1033.022,312.549,-124.978,171.479,44.984,158.704
C05932=1033.014,312.301,-124.944,171.474,44.984,158.703
C05933=1033.007,312.054,-124.910,171.469,44.983,158.703
C05934=1033.001,311.806,-124.876,171.464,44.982,158.702
C05935=1032.994,311.559,-124.843,171.460,44.981,158.701
C05936=1032.987,311.311,-124.809,171.456,44.980,158.701
C05937=1032.980,311.063,-124.775,171.451,44.979,158.700
C05938=1032.973,310.816,-124.741,171.447,44.979,158.700
C05939=1032.965,310.568,-124.707,171.442,44.978,158.699
C05940=1032.958,310.321,-124.674,171.437,44.978,158.698
C05941=1032.951,310.073,-124.641,171.433,44.977,158.698
C05942=1032.944,309.825,-124.607,171.428,44.976,158.697
C05943=1032.937,309.578,-124.574,171.423,44.975,158.696
C05944=1032.929,309.330,-124.540,171.419,44.975,158.696
C05945=1032.922,309.083,-124.507,171.415,44.974,158.695
C05946=1032.915,308.835,-124.474,171.410,44.973,158.695
C05947=1032.908,308.587,-124.440,171.405,44.973,158.694
C05948=1032.901,308.340,-124.406,171.401,44.972,158.693
C05949=1032.894,308.092,-124.374,171.396,44.971,158.693
C05950=1032.887,307.845,-124.340,171.392,44.971,158.692
C05951=1032.879,307.597,-124.306,171.387,44.971,158.692
C05952=1032.873,307.349,-124.273,171.383,44.969,158.691
C05953=1032.865,307.102,-124.240,171.379,44.969,158.690
C05954=1032.854,306.710,-124.188,171.372,44.968,158.690
C05955=1032.843,306.318,-124.134,171.364,44.967,158.689
C05956=1032.832,305.927,-124.082,171.358,44.966,158.688
C05957=1032.820,305.536,-124.029,171.351,44.965,158.687
C05958=1032.814,305.287,-123.996,171.346,44.964,158.686
C05959=1032.807,305.041,-123.963,171.341,44.964,158.686
C05960=1032.799,304.793,-123.930,171.337,44.964,158.685
C05961=1032.793,304.546,-123.897,171.332,44.963,158.685
C05962=1032.786,304.297,-123.864,171.328,44.962,158.684
C05963=1032.779,304.049,-123.831,171.324,44.962,158.683
C05964=1032.772,303.802,-123.798,171.319,44.961,158.683
C05965=1032.765,303.554,-123.765,171.314,44.960,158.682
C05966=1032.758,303.307,-123.731,171.311,44.960,158.682
C05967=1032.751,303.059,-123.698,171.306,44.959,158.681
C05968=1032.744,302.811,-123.666,171.302,44.959,158.681
C05969=1032.737,302.564,-123.632,171.297,44.958,158.680
C05970=1032.731,302.316,-123.599,171.293,44.958,158.679
C05971=1032.724,302.068,-123.566,171.289,44.957,158.679
C05972=1032.716,301.821,-123.533,171.284,44.957,158.678
C05973=1032.710,301.573,-123.500,171.280,44.957,158.678
C05974=1032.703,301.325,-123.467,171.276,44.955,158.677
C05975=1032.696,301.078,-123.434,171.271,44.955,158.677
C05976=1032.689,300.830,-123.401,171.267,44.955,158.676
C05977=1032.682,300.582,-123.368,171.263,44.954,158.676
C05978=1032.676,300.335,-123.336,171.259,44.954,158.675
C05979=1032.668,300.087,-123.302,171.254,44.953,158.674
C05980=1032.662,299.840,-123.270,171.249,44.952,158.674
C05981=1032.655,299.591,-123.237,171.246,44.952,158.673
C05982=1032.648,299.344,-123.204,171.241,44.952,158.673
C05983=1032.641,299.096,-123.171,171.237,44.951,158.672
C05984=1032.634,298.848,-123.139,171.233,44.951,158.672
C05985=1032.628,298.600,-123.106,171.229,44.950,158.671
C05986=1032.621,298.353,-123.072,171.224,44.950,158.671
C05987=1032.614,298.106,-123.040,171.221,44.949,158.670
C05988=1032.607,297.857,-123.007,171.216,44.948,158.670
C05989=1032.601,297.610,-122.974,171.211,44.948,158.669
C05990=1032.594,297.362,-122.942,171.208,44.947,158.669
C05991=1032.587,297.114,-122.909,171.203,44.947,158.668
C05992=1032.581,296.866,-122.876,171.199,44.947,158.667
C05993=1032.574,296.619,-122.844,171.195,44.946,158.667
C05994=1032.567,296.371,-122.811,171.190,44.946,158.666
C05995=1032.560,296.123,-122.778,171.187,44.945,158.666
C05996=1032.554,295.876,-122.745,171.182,44.945,158.665
C05997=1032.547,295.628,-122.713,171.178,44.945,158.665
C05998=1032.540,295.380,-122.680,171.174,44.944,158.664
C05999=1032.534,295.133,-122.647,171.170,44.944,158.664
C06000=1032.527,294.885,-122.615,171.165,44.943,158.663
C06001=1032.520,294.636,-122.583,171.162,44.943,158.663
C06002=1032.513,294.389,-122.551,171.157,44.942,158.662
C06003=1032.507,294.141,-122.518,171.153,44.942,158.662
C06004=1032.499,293.893,-122.485,171.149,44.942,158.661
C06005=1032.493,293.645,-122.453,171.145,44.942,158.661
C06006=1032.486,293.398,-122.421,171.141,44.941,158.660
C06007=1032.479,293.151,-122.389,171.137,44.941,158.660
C06008=1032.473,292.902,-122.357,171.132,44.940,158.659
C06009=1032.466,292.655,-122.324,171.129,44.940,158.659
C06010=1032.455,292.280,-122.275,171.122,44.940,158.658
C06011=1032.445,291.906,-122.227,171.116,44.939,158.658
C06012=1032.434,291.531,-122.179,171.110,44.939,158.657
C06013=1032.424,291.157,-122.130,171.104,44.939,158.656
C06014=1032.417,290.908,-122.098,171.099,44.938,158.656
C06015=1032.410,290.661,-122.066,171.096,44.938,158.655
C06016=1032.404,290.413,-122.034,171.091,44.938,158.655
C06017=1032.397,290.165,-122.002,171.088,44.937,158.654
C06018=1032.390,289.917,-121.970,171.083,44.938,158.654
C06019=1032.383,289.669,-121.939,171.079,44.937,158.653
C06020=1032.377,289.421,-121.906,171.075,44.937,158.653
C06021=1032.370,289.173,-121.874,171.071,44.937,158.653
C06022=1032.363,288.926,-121.842,171.068,44.936,158.652
C06023=1032.356,288.678,-121.811,171.063,44.936,158.652
C06024=1032.349,288.430,-121.779,171.060,44.936,158.651
C06025=1032.342,288.182,-121.747,171.055,44.936,158.651
C06026=1032.336,287.934,-121.715,171.051,44.936,158.650
C06027=1032.329,287.686,-121.684,171.047,44.935,158.650
C06028=1032.322,287.439,-121.651,171.043,44.936,158.649
C06029=1032.315,287.191,-121.620,171.039,44.935,158.649
C06030=1032.309,286.943,-121.588,171.035,44.935,158.648
C06031=1032.301,286.695,-121.556,171.032,44.935,158.648
C06032=1032.295,286.447,-121.524,171.027,44.934,158.648
C06033=1032.288,286.199,-121.493,171.024,44.934,158.647
C06034=1032.281,285.951,-121.461,171.019,44.934,158.647
C06035=1032.275,285.703,-121.430,171.016,44.934,158.646
C06036=1032.268,285.456,-121.398,171.012,44.934,158.646
C06037=1032.260,285.208,-121.367,171.007,44.934,158.646
C06038=1032.254,284.960,-121.335,171.004,44.934,158.645
C06039=1032.247,284.713,-121.304,170.999,44.934,158.645
C06040=1032.240,284.465,-121.272,170.996,44.934,158.644
C06041=1032.233,284.216,-121.241,170.991,44.933,158.644
C06042=1032.226,283.968,-121.209,170.988,44.933,158.644
C06043=1032.219,283.720,-121.178,170.984,44.934,158.643
C06044=1032.213,283.472,-121.146,170.980,44.933,158.643
C06045=1032.206,283.224,-121.115,170.976,44.933,158.642
C06046=1032.199,282.977,-121.083,170.973,44.933,158.642
C06047=1032.192,282.729,-121.052,170.968,44.933,158.641
C06048=1032.186,282.481,-121.021,170.965,44.933,158.641
C06049=1032.179,282.233,-120.989,170.960,44.933,158.641
C06050=1032.172,281.985,-120.958,170.957,44.933,158.640
C06051=1032.166,281.737,-120.926,170.953,44.933,158.640
C06052=1032.158,281.489,-120.895,170.949,44.932,158.639
C06053=1032.151,281.242,-120.864,170.945,44.933,158.639
C06054=1032.145,280.994,-120.833,170.942,44.933,158.639
C06055=1032.138,280.745,-120.802,170.937,44.932,158.638
C06056=1032.131,280.497,-120.770,170.934,44.932,158.638
C06057=1032.125,280.249,-120.739,170.929,44.933,158.638
C06058=1032.118,280.001,-120.708,170.926,44.933,158.637
C06059=1032.111,279.754,-120.676,170.922,44.932,158.637
C06060=1032.105,279.506,-120.645,170.918,44.932,158.636
C06061=1032.099,279.258,-120.614,170.914,44.933,158.636
C06062=1032.092,279.010,-120.583,170.911,44.932,158.636
C06063=1032.085,278.762,-120.551,170.907,44.932,158.635
C06064=1032.078,278.514,-120.521,170.903,44.932,158.635
C06065=1032.071,278.266,-120.489,170.900,44.932,158.635
C06066=1032.062,277.903,-120.443,170.894,44.932,158.634
C06067=1032.052,277.541,-120.398,170.889,44.932,158.633
C06068=1032.042,277.178,-120.353,170.883,44.933,158.633
C06069=1032.032,276.816,-120.308,170.878,44.933,158.632
C06070=1032.025,276.568,-120.278,170.873,44.933,158.632
C06071=1032.018,276.320,-120.246,170.870,44.933,158.632
C06072=1032.012,276.072,-120.215,170.866,44.933,158.631
C06073=1032.004,275.824,-120.185,170.862,44.933,158.631
C06074=1031.999,275.576,-120.154,170.858,44.933,158.630
C06075=1031.992,275.329,-120.123,170.855,44.933,158.630
C06076=1031.985,275.080,-120.093,170.851,44.933,158.630
C06077=1031.978,274.832,-120.061,170.847,44.933,158.629
C06078=1031.971,274.584,-120.030,170.844,44.933,158.629
C06079=1031.964,274.336,-120.000,170.839,44.933,158.629
C06080=1031.958,274.088,-119.969,170.836,44.933,158.628
C06081=1031.951,273.841,-119.938,170.832,44.934,158.628
C06082=1031.944,273.592,-119.908,170.829,44.934,158.628
C06083=1031.938,273.344,-119.877,170.825,44.934,158.627
C06084=1031.930,273.096,-119.846,170.821,44.934,158.627
C06085=1031.925,272.848,-119.816,170.818,44.934,158.627
C06086=1031.918,272.600,-119.785,170.813,44.934,158.626
C06087=1031.911,272.352,-119.754,170.810,44.934,158.626
C06088=1031.904,272.104,-119.724,170.807,44.934,158.626
C06089=1031.897,271.856,-119.693,170.803,44.935,158.625
C06090=1031.891,271.608,-119.662,170.799,44.935,158.625
C06091=1031.884,271.360,-119.632,170.796,44.935,158.625
C06092=1031.877,271.112,-119.602,170.792,44.935,158.624
C06093=1031.871,270.864,-119.570,170.788,44.935,158.624
C06094=1031.864,270.616,-119.540,170.784,44.935,158.624
C06095=1031.858,270.368,-119.510,170.781,44.935,158.623
C06096=1031.851,270.119,-119.479,170.778,44.935,158.623
C06097=1031.844,269.872,-119.450,170.773,44.936,158.623
C06098=1031.837,269.624,-119.418,170.770,44.936,158.623
C06099=1031.830,269.376,-119.388,170.767,44.936,158.622
C06100=1031.824,269.127,-119.357,170.763,44.937,158.622
C06101=1031.817,268.880,-119.328,170.759,44.937,158.621
C06102=1031.810,268.632,-119.298,170.756,44.937,158.621
C06103=1031.804,268.383,-119.267,170.752,44.937,158.621
C06104=1031.797,268.136,-119.237,170.748,44.937,158.620
C06105=1031.791,267.887,-119.206,170.744,44.938,158.620
C06106=1031.784,267.639,-119.176,170.741,44.938,158.620
C06107=1031.777,267.391,-119.147,170.738,44.938,158.620
C06108=1031.771,267.143,-119.116,170.734,44.938,158.619
C06109=1031.763,266.895,-119.086,170.730,44.938,158.619
C06110=1031.758,266.647,-119.055,170.727,44.939,158.619
C06111=1031.750,266.399,-119.025,170.723,44.939,158.618
C06112=1031.743,266.150,-118.995,170.720,44.939,158.618
C06113=1031.737,265.903,-118.965,170.716,44.939,158.618
C06114=1031.730,265.654,-118.935,170.712,44.940,158.618
C06115=1031.723,265.406,-118.904,170.709,44.940,158.617
C06116=1031.717,265.159,-118.875,170.706,44.940,158.617
C06117=1031.709,264.910,-118.845,170.701,44.940,158.617
C06118=1031.704,264.663,-118.814,170.698,44.941,158.616
C06119=1031.696,264.414,-118.784,170.695,44.941,158.616
C06120=1031.690,264.165,-118.755,170.691,44.941,158.616
C06121=1031.683,263.918,-118.725,170.688,44.942,158.616
C06122=1031.673,263.560,-118.681,170.682,44.943,158.615
C06123=1031.664,263.202,-118.638,170.678,44.943,158.615
C06124=1031.654,262.844,-118.595,170.673,44.943,158.614
C06125=1031.645,262.487,-118.551,170.668,44.944,158.614
C06126=1031.638,262.238,-118.522,170.664,44.944,158.614
C06127=1031.631,261.990,-118.492,170.661,44.944,158.613
C06128=1031.624,261.742,-118.462,170.657,44.945,158.613
C06129=1031.618,261.494,-118.431,170.654,44.945,158.613
C06130=1031.612,261.246,-118.402,170.650,44.945,158.612
C06131=1031.605,260.998,-118.372,170.646,44.946,158.612
C06132=1031.598,260.749,-118.343,170.643,44.946,158.612
C06133=1031.590,260.501,-118.314,170.640,44.946,158.612
C06134=1031.584,260.253,-118.285,170.636,44.947,158.611
C06135=1031.577,260.005,-118.254,170.633,44.947,158.611
C06136=1031.570,259.756,-118.225,170.630,44.948,158.611
C06137=1031.564,259.509,-118.195,170.625,44.948,158.611
C06138=1031.557,259.260,-118.166,170.622,44.949,158.611
C06139=1031.549,259.013,-118.137,170.619,44.949,158.610
C06140=1031.543,258.764,-118.107,170.616,44.950,158.610
C06141=1031.536,258.516,-118.078,170.612,44.950,158.610
C06142=1031.529,258.268,-118.048,170.609,44.951,158.610
C06143=1031.523,258.020,-118.018,170.606,44.951,158.609
C06144=1031.516,257.771,-117.989,170.601,44.951,158.609
C06145=1031.509,257.524,-117.960,170.598,44.952,158.609
C06146=1031.502,257.275,-117.930,170.595,44.952,158.609
C06147=1031.495,257.027,-117.901,170.592,44.953,158.608
C06148=1031.488,256.779,-117.871,170.588,44.953,158.608
C06149=1031.482,256.531,-117.842,170.585,44.954,158.608
C06150=1031.475,256.282,-117.813,170.582,44.954,158.608
C06151=1031.468,256.035,-117.784,170.577,44.955,158.607
C06152=1031.461,255.786,-117.754,170.574,44.955,158.607
C06153=1031.455,255.538,-117.725,170.571,44.956,158.607
C06154=1031.448,255.290,-117.695,170.568,44.956,158.607
C06155=1031.441,255.041,-117.666,170.564,44.957,158.606
C06156=1031.435,254.793,-117.637,170.561,44.957,158.606
C06157=1031.428,254.545,-117.608,170.558,44.958,158.606
C06158=1031.421,254.297,-117.578,170.554,44.958,158.606
C06159=1031.414,254.048,-117.549,170.551,44.958,158.606
C06160=1031.408,253.800,-117.520,170.547,44.959,158.605
C06161=1031.402,253.552,-117.491,170.544,44.960,158.605
C06162=1031.394,253.304,-117.461,170.541,44.960,158.605
C06163=1031.387,253.056,-117.432,170.538,44.961,158.605
C06164=1031.381,252.808,-117.403,170.534,44.961,158.604
C06165=1031.374,252.559,-117.374,170.530,44.961,158.604
C06166=1031.368,252.311,-117.345,170.527,44.962,158.604
C06167=1031.361,252.063,-117.315,170.524,44.963,158.604
C06168=1031.354,251.815,-117.286,170.521,44.963,158.604
C06169=1031.348,251.567,-117.257,170.517,44.964,158.603
C06170=1031.341,251.318,-117.228,170.514,44.964,158.603
C06171=1031.335,251.070,-117.199,170.511,44.964,158.603
C06172=1031.328,250.822,-117.170,170.508,44.965,158.603
C06173=1031.321,250.574,-117.141,170.505,44.966,158.603
C06174=1031.315,250.325,-117.112,170.500,44.966,158.602
C06175=1031.308,250.078,-117.082,170.497,44.967,158.602
C06176=1031.302,249.829,-117.053,170.494,44.967,158.602
C06177=1031.295,249.581,-117.024,170.491,44.968,158.602
C06178=1031.286,249.222,-116.983,170.486,44.968,158.601
C06179=1031.276,248.863,-116.940,170.482,44.969,158.601
C06180=1031.267,248.503,-116.898,170.477,44.970,158.601
C06181=1031.257,248.144,-116.856,170.473,44.971,158.600
C06182=1031.250,247.896,-116.827,170.468,44.972,158.600
C06183=1031.244,247.648,-116.798,170.465,44.972,158.600
C06184=1031.237,247.399,-116.769,170.462,44.972,158.600
C06185=1031.230,247.151,-116.740,170.459,44.973,158.600
C06186=1031.224,246.903,-116.711,170.456,44.974,158.599
C06187=1031.218,246.655,-116.682,170.453,44.974,158.599
C06188=1031.212,246.406,-116.654,170.450,44.974,158.599
C06189=1031.204,246.157,-116.625,170.447,44.975,158.599
C06190=1031.198,245.909,-116.596,170.443,44.976,158.599
C06191=1031.192,245.661,-116.567,170.439,44.976,158.598
C06192=1031.186,245.413,-116.538,170.436,44.977,158.598
C06193=1031.179,245.165,-116.509,170.433,44.977,158.598
C06194=1031.172,244.917,-116.480,170.430,44.978,158.598
C06195=1031.165,244.668,-116.451,170.427,44.979,158.598
C06196=1031.159,244.419,-116.423,170.424,44.979,158.597
C06197=1031.152,244.172,-116.394,170.421,44.979,158.597
C06198=1031.146,243.923,-116.365,170.418,44.980,158.597
C06199=1031.139,243.676,-116.337,170.414,44.981,158.597
C06200=1031.133,243.427,-116.308,170.411,44.982,158.597
C06201=1031.126,243.178,-116.280,170.408,44.982,158.596
C06202=1031.119,242.930,-116.251,170.405,44.983,158.596
C06203=1031.113,242.682,-116.223,170.402,44.984,158.596
C06204=1031.107,242.434,-116.194,170.399,44.984,158.596
C06205=1031.100,242.186,-116.165,170.396,44.985,158.596
C06206=1031.094,241.937,-116.137,170.393,44.986,158.596
C06207=1031.086,241.689,-116.108,170.388,44.986,158.595
C06208=1031.080,241.440,-116.079,170.385,44.986,158.595
C06209=1031.073,241.192,-116.052,170.382,44.987,158.595
C06210=1031.067,240.944,-116.022,170.379,44.988,158.595
C06211=1031.060,240.695,-115.995,170.376,44.988,158.595
C06212=1031.054,240.447,-115.966,170.373,44.989,158.594
C06213=1031.047,240.199,-115.937,170.370,44.990,158.594
C06214=1031.041,239.951,-115.909,170.367,44.990,158.594
C06215=1031.034,239.703,-115.880,170.364,44.991,158.594
C06216=1031.027,239.454,-115.852,170.360,44.992,158.594
C06217=1031.020,239.205,-115.825,170.357,44.993,158.594
C06218=1031.014,238.957,-115.796,170.354,44.994,158.594
C06219=1031.007,238.709,-115.768,170.351,44.995,158.593
C06220=1031.000,238.461,-115.739,170.348,44.995,158.593
C06221=1030.993,238.212,-115.712,170.345,44.996,158.593
C06222=1030.987,237.964,-115.683,170.342,44.997,158.593
C06223=1030.981,237.716,-115.655,170.339,44.997,158.593
C06224=1030.974,237.467,-115.627,170.336,44.998,158.593
C06225=1030.967,237.220,-115.599,170.333,44.999,158.592
C06226=1030.960,236.970,-115.570,170.329,45.000,158.592
C06227=1030.954,236.722,-115.542,170.326,45.000,158.592
C06228=1030.947,236.474,-115.514,170.323,45.001,158.592
C06229=1030.940,236.225,-115.486,170.320,45.002,158.592
C06230=1030.933,235.977,-115.458,170.317,45.003,158.592
C06231=1030.927,235.729,-115.429,170.314,45.003,158.592
C06232=1030.920,235.480,-115.402,170.311,45.004,158.591
C06233=1030.914,235.232,-115.374,170.308,45.005,158.591
C06234=1030.904,234.866,-115.333,170.303,45.006,158.591
C06235=1030.894,234.502,-115.291,170.299,45.007,158.591
C06236=1030.884,234.136,-115.250,170.294,45.009,158.591
C06237=1030.874,233.771,-115.209,170.290,45.009,158.590
C06238=1030.869,233.523,-115.181,170.287,45.010,158.590
C06239=1030.862,233.275,-115.153,170.284,45.011,158.590
C06240=1030.855,233.027,-115.125,170.281,45.012,158.590
C06241=1030.848,232.778,-115.098,170.278,45.013,158.590
C06242=1030.842,232.530,-115.070,170.275,45.013,158.590
C06243=1030.835,232.281,-115.042,170.272,45.014,158.590
C06244=1030.829,232.033,-115.013,170.268,45.015,158.589
C06245=1030.822,231.785,-114.985,170.265,45.016,158.589
C06246=1030.815,231.536,-114.958,170.262,45.017,158.589
C06247=1030.809,231.288,-114.930,170.259,45.018,158.589
C06248=1030.802,231.039,-114.902,170.256,45.018,158.589
C06249=1030.795,230.791,-114.874,170.253,45.019,158.589
C06250=1030.789,230.542,-114.847,170.250,45.020,158.589
C06251=1030.782,230.294,-114.819,170.247,45.021,158.589
C06252=1030.775,230.046,-114.791,170.244,45.022,158.589
C06253=1030.769,229.797,-114.763,170.241,45.023,158.589
C06254=1030.762,229.549,-114.736,170.238,45.024,158.588
C06255=1030.755,229.300,-114.708,170.235,45.024,158.588
C06256=1030.749,229.052,-114.680,170.232,45.025,158.588
C06257=1030.743,228.804,-114.653,170.229,45.026,158.588
C06258=1030.736,228.556,-114.625,170.226,45.027,158.588
C06259=1030.729,228.307,-114.597,170.223,45.028,158.588
C06260=1030.723,228.059,-114.570,170.221,45.029,158.588
C06261=1030.716,227.810,-114.542,170.218,45.029,158.588
C06262=1030.709,227.562,-114.514,170.214,45.030,158.587
C06263=1030.702,227.313,-114.487,170.212,45.031,158.587
C06264=1030.696,227.064,-114.460,170.209,45.032,158.587
C06265=1030.689,226.816,-114.432,170.206,45.033,158.587
C06266=1030.683,226.568,-114.405,170.203,45.034,158.587
C06267=1030.676,226.320,-114.377,170.200,45.035,158.587
C06268=1030.669,226.072,-114.350,170.197,45.036,158.587
C06269=1030.663,225.823,-114.322,170.194,45.037,158.587
C06270=1030.655,225.574,-114.295,170.191,45.037,158.587
C06271=1030.649,225.326,-114.268,170.188,45.039,158.587
C06272=1030.642,225.078,-114.240,170.185,45.039,158.586
C06273=1030.635,224.829,-114.212,170.182,45.041,158.586
C06274=1030.629,224.581,-114.186,170.179,45.041,158.586
C06275=1030.622,224.333,-114.158,170.177,45.043,158.586
C06276=1030.616,224.084,-114.131,170.173,45.043,158.586
C06277=1030.609,223.835,-114.104,170.170,45.044,158.586
C06278=1030.602,223.587,-114.076,170.168,45.045,158.586
C06279=1030.595,223.339,-114.049,170.165,45.046,158.586
C06280=1030.589,223.091,-114.021,170.162,45.047,158.586
C06281=1030.583,222.842,-113.994,170.159,45.048,158.586
C06282=1030.576,222.593,-113.967,170.156,45.049,158.586
C06283=1030.568,222.345,-113.940,170.153,45.050,158.585
C06284=1030.562,222.096,-113.913,170.150,45.051,158.585
C06285=1030.556,221.848,-113.885,170.147,45.052,158.585
C06286=1030.550,221.599,-113.858,170.144,45.053,158.585
C06287=1030.542,221.351,-113.831,170.141,45.054,158.585
C06288=1030.536,221.103,-113.803,170.138,45.055,158.585
C06289=1030.529,220.854,-113.776,170.136,45.056,158.585
C06290=1030.519,220.481,-113.735,170.131,45.058,158.585
C06291=1030.509,220.109,-113.695,170.127,45.059,158.585
C06292=1030.500,219.736,-113.654,170.123,45.060,158.585
C06293=1030.490,219.362,-113.613,170.118,45.062,158.584
C06294=1030.483,219.115,-113.586,170.115,45.062,158.584
C06295=1030.477,218.866,-113.559,170.112,45.064,158.584
C06296=1030.469,218.618,-113.532,170.109,45.064,158.584
C06297=1030.463,218.368,-113.505,170.106,45.066,158.584
C06298=1030.456,218.121,-113.478,170.104,45.067,158.584
C06299=1030.450,217.872,-113.451,170.101,45.068,158.584
C06300=1030.443,217.623,-113.425,170.098,45.069,158.584
C06301=1030.436,217.375,-113.397,170.095,45.070,158.584
C06302=1030.429,217.127,-113.371,170.092,45.071,158.584
C06303=1030.423,216.878,-113.343,170.089,45.072,158.584
C06304=1030.416,216.630,-113.317,170.086,45.073,158.584
C06305=1030.410,216.381,-113.290,170.084,45.074,158.584
C06306=1030.402,216.133,-113.263,170.082,45.075,158.584
C06307=1030.395,215.884,-113.237,170.079,45.076,158.583
C06308=1030.389,215.635,-113.210,170.076,45.077,158.583
C06309=1030.382,215.388,-113.183,170.073,45.078,158.583
C06310=1030.376,215.139,-113.156,170.070,45.079,158.583
C06311=1030.369,214.890,-113.130,170.067,45.081,158.583
C06312=1030.363,214.642,-113.103,170.064,45.081,158.583
C06313=1030.355,214.393,-113.076,170.061,45.083,158.583
C06314=1030.349,214.144,-113.049,170.059,45.084,158.583
C06315=1030.343,213.896,-113.023,170.056,45.085,158.583
C06316=1030.336,213.648,-112.995,170.053,45.086,158.583
C06317=1030.329,213.399,-112.969,170.050,45.087,158.583
C06318=1030.323,213.151,-112.942,170.047,45.088,158.583
C06319=1030.316,212.902,-112.915,170.044,45.089,158.583
C06320=1030.310,212.654,-112.888,170.042,45.090,158.583
C06321=1030.303,212.406,-112.862,170.039,45.091,158.583
C06322=1030.296,212.157,-112.835,170.037,45.092,158.583
C06323=1030.290,211.908,-112.809,170.034,45.094,158.583
C06324=1030.283,211.660,-112.782,170.031,45.094,158.583
C06325=1030.277,211.412,-112.755,170.028,45.096,158.582
C06326=1030.269,211.163,-112.728,170.025,45.096,158.582
C06327=1030.263,210.914,-112.701,170.022,45.098,158.582
C06328=1030.257,210.666,-112.675,170.019,45.099,158.582
C06329=1030.249,210.417,-112.649,170.017,45.100,158.582
C06330=1030.244,210.169,-112.622,170.014,45.101,158.582
C06331=1030.237,209.920,-112.596,170.012,45.102,158.582
C06332=1030.229,209.672,-112.569,170.009,45.103,158.582
C06333=1030.223,209.423,-112.543,170.006,45.105,158.582
C06334=1030.217,209.174,-112.516,170.003,45.105,158.582
C06335=1030.210,208.926,-112.490,170.000,45.107,158.582
C06336=1030.203,208.678,-112.464,169.998,45.108,158.582
C06337=1030.196,208.429,-112.437,169.995,45.109,158.582
C06338=1030.190,208.180,-112.411,169.992,45.110,158.582
C06339=1030.183,207.932,-112.384,169.989,45.111,158.582
C06340=1030.176,207.684,-112.358,169.986,45.112,158.582
C06341=1030.169,207.435,-112.332,169.984,45.114,158.582
C06342=1030.163,207.187,-112.306,169.982,45.115,158.582
C06343=1030.156,206.938,-112.279,169.979,45.116,158.582
C06344=1030.150,206.690,-112.253,169.976,45.117,158.582
C06345=1030.143,206.441,-112.226,169.973,45.118,158.582
C06346=1030.133,206.074,-112.187,169.969,45.120,158.582
C06347=1030.123,205.707,-112.149,169.965,45.122,158.582
C06348=1030.113,205.340,-112.110,169.961,45.124,158.582
C06349=1030.102,204.973,-112.071,169.957,45.125,158.582
C06350=1030.073,203.714,-111.946,169.595,45.023,158.524
C06351=1030.062,203.294,-111.904,169.589,45.027,158.524
C06352=1030.056,203.046,-111.879,169.585,45.028,158.524
C06353=1030.050,202.797,-111.855,169.582,45.031,158.524
C06354=1030.044,202.549,-111.830,169.578,45.033,158.524
C06355=1030.038,202.300,-111.805,169.574,45.034,158.524
C06356=1030.033,202.052,-111.780,169.571,45.037,158.524
C06357=1030.027,201.802,-111.755,169.567,45.039,158.524
C06358=1030.020,201.554,-111.730,169.563,45.040,158.524
C06359=1030.014,201.305,-111.706,169.559,45.043,158.524
C06360=1030.008,201.057,-111.681,169.555,45.045,158.524
C06361=1030.002,200.807,-111.656,169.551,45.046,158.524
C06362=1029.997,200.559,-111.632,169.548,45.048,158.524
C06363=1029.991,200.310,-111.607,169.544,45.051,158.524
C06364=1029.984,200.061,-111.583,169.541,45.053,158.524
C06365=1029.979,199.813,-111.558,169.537,45.055,158.525
C06366=1029.972,199.564,-111.534,169.533,45.057,158.524
C06367=1029.966,199.315,-111.509,169.530,45.059,158.525
C06368=1029.960,199.067,-111.485,169.526,45.061,158.525
C06369=1029.954,198.817,-111.461,169.523,45.063,158.525
C06370=1029.947,198.569,-111.436,169.519,45.065,158.525
C06371=1029.942,198.320,-111.412,169.516,45.067,158.525
C06372=1029.935,198.071,-111.388,169.512,45.070,158.525
C06373=1029.929,197.822,-111.363,169.508,45.072,158.525
C06374=1029.923,197.574,-111.340,169.505,45.074,158.525
C06375=1029.917,197.325,-111.314,169.501,45.076,158.525
C06376=1029.911,197.077,-111.291,169.498,45.078,158.525
C06377=1029.905,196.828,-111.266,169.494,45.080,158.525
C06378=1029.898,196.579,-111.242,169.490,45.082,158.525
C06379=1029.893,196.330,-111.218,169.487,45.084,158.525
C06380=1029.887,196.081,-111.194,169.483,45.086,158.526
C06381=1029.880,195.833,-111.170,169.480,45.089,158.526
C06382=1029.874,195.584,-111.145,169.476,45.091,158.526
C06383=1029.868,195.336,-111.121,169.473,45.093,158.526
C06384=1029.862,195.087,-111.096,169.469,45.095,158.526
C06385=1029.856,194.838,-111.073,169.466,45.097,158.526
C06386=1029.850,194.589,-111.048,169.462,45.100,158.526
C06387=1029.844,194.340,-111.024,169.459,45.102,158.526
C06388=1029.838,194.091,-111.000,169.455,45.104,158.526
C06389=1029.832,193.842,-110.976,169.451,45.106,158.526
C06390=1029.827,193.594,-110.951,169.448,45.108,158.526
C06391=1029.820,193.345,-110.927,169.444,45.110,158.526
C06392=1029.815,193.096,-110.903,169.441,45.112,158.526
C06393=1029.809,192.848,-110.880,169.437,45.114,158.527
C06394=1029.802,192.599,-110.855,169.433,45.116,158.527
C06395=1029.797,192.350,-110.831,169.430,45.119,158.527
C06396=1029.790,192.101,-110.807,169.426,45.121,158.527
C06397=1029.785,191.853,-110.783,169.423,45.123,158.527
C06398=1029.778,191.604,-110.759,169.419,45.125,158.527
C06399=1029.773,191.355,-110.735,169.416,45.127,158.527
C06400=1029.765,191.015,-110.702,169.411,45.130,158.527
C06401=1029.756,190.675,-110.670,169.406,45.134,158.527
C06402=1029.748,190.335,-110.637,169.401,45.136,158.527
C06403=1029.740,189.995,-110.604,169.397,45.139,158.528
C06404=1029.735,189.746,-110.580,169.394,45.141,158.528
C06405=1029.728,189.498,-110.556,169.390,45.144,158.528
C06406=1029.722,189.249,-110.532,169.386,45.146,158.528
C06407=1029.717,189.000,-110.508,169.383,45.148,158.528
C06408=1029.710,188.716,-110.481,169.379,45.150,158.528
C06409=1029.703,188.433,-110.454,169.375,45.153,158.528
C06410=1029.696,188.150,-110.426,169.371,45.155,158.528
C06411=1029.690,187.866,-110.399,169.367,45.158,158.528
C06412=1029.684,187.618,-110.376,169.364,45.160,158.528
C06413=1029.678,187.369,-110.351,169.361,45.162,158.529
C06414=1029.672,187.120,-110.327,169.357,45.164,158.529
C06415=1029.666,186.871,-110.304,169.354,45.166,158.529
C06416=1029.660,186.622,-110.280,169.350,45.169,158.529
C06417=1029.654,186.374,-110.256,169.347,45.171,158.529
C06418=1029.649,186.125,-110.233,169.343,45.174,158.529
C06419=1029.643,185.876,-110.209,169.341,45.176,158.529
C06420=1029.637,185.627,-110.184,169.337,45.178,158.529
C06421=1029.632,185.378,-110.161,169.334,45.180,158.529
C06422=1029.626,185.130,-110.138,169.330,45.182,158.530
C06423=1029.620,184.881,-110.113,169.327,45.184,158.530
C06424=1029.614,184.632,-110.090,169.323,45.187,158.530
C06425=1029.609,184.383,-110.066,169.321,45.188,158.530
C06426=1029.603,184.135,-110.042,169.317,45.191,158.530
C06427=1029.596,183.885,-110.019,169.313,45.193,158.530
C06428=1029.591,183.637,-109.995,169.310,45.195,158.530
C06429=1029.585,183.388,-109.971,169.306,45.197,158.530
C06430=1029.580,183.139,-109.947,169.304,45.199,158.530
C06431=1029.573,182.890,-109.923,169.300,45.201,158.530
C06432=1029.568,182.641,-109.900,169.297,45.204,158.530
C06433=1029.562,182.392,-109.877,169.293,45.207,158.531
C06434=1029.555,182.143,-109.853,169.290,45.209,158.531
C06435=1029.549,181.895,-109.831,169.287,45.212,158.531
C06436=1029.543,181.647,-109.807,169.283,45.214,158.531
C06437=1029.537,181.398,-109.785,169.279,45.216,158.531
C06438=1029.531,181.148,-109.761,169.277,45.219,158.532
C06439=1029.525,180.899,-109.738,169.274,45.221,158.532
C06440=1029.518,180.651,-109.715,169.270,45.223,158.532
C06441=1029.512,180.402,-109.692,169.267,45.226,158.532
C06442=1029.506,180.153,-109.669,169.263,45.228,158.532
C06443=1029.500,179.904,-109.645,169.260,45.231,158.532
C06444=1029.494,179.656,-109.622,169.256,45.233,158.532
C06445=1029.487,179.406,-109.600,169.253,45.235,158.532
C06446=1029.482,179.157,-109.577,169.251,45.238,158.533
C06447=1029.476,178.908,-109.554,169.247,45.240,158.533
C06448=1029.470,178.660,-109.530,169.244,45.243,158.533
C06449=1029.464,178.411,-109.507,169.240,45.245,158.533
C06450=1029.457,178.162,-109.484,169.237,45.247,158.533
C06451=1029.451,177.913,-109.461,169.233,45.250,158.533
C06452=1029.446,177.664,-109.438,169.230,45.252,158.534
C06453=1029.439,177.416,-109.415,169.227,45.254,158.534
C06454=1029.434,177.167,-109.392,169.224,45.257,158.534
C06455=1029.427,176.918,-109.369,169.220,45.260,158.534
C06456=1029.421,176.669,-109.346,169.217,45.262,158.534
C06457=1029.415,176.420,-109.323,169.214,45.265,158.534
C06458=1029.409,176.171,-109.300,169.211,45.267,158.535
C06459=1029.404,175.922,-109.277,169.208,45.269,158.535
C06460=1029.397,175.674,-109.254,169.204,45.272,158.535
C06461=1029.391,175.425,-109.231,169.201,45.274,158.535
C06462=1029.385,175.176,-109.208,169.197,45.277,158.535
C06463=1029.379,174.927,-109.185,169.195,45.279,158.535
C06464=1029.373,174.678,-109.163,169.191,45.282,158.535
C06465=1029.367,174.429,-109.140,169.188,45.284,158.536
C06466=1029.361,174.180,-109.117,169.185,45.287,158.536
C06467=1029.356,173.932,-109.094,169.181,45.289,158.536
C06468=1029.350,173.683,-109.071,169.179,45.291,158.536
C06469=1029.343,173.433,-109.048,169.175,45.294,158.536
C06470=1029.337,173.184,-109.025,169.172,45.296,158.536
C06471=1029.331,172.936,-109.002,169.168,45.299,158.537
C06472=1029.325,172.652,-108.976,169.165,45.302,158.537
C06473=1029.318,172.368,-108.951,169.162,45.304,158.537
C06474=1029.311,172.085,-108.925,169.157,45.307,158.537
C06475=1029.304,171.801,-108.898,169.154,45.310,158.537
C06476=1029.298,171.552,-108.875,169.150,45.312,158.537
C06477=1029.293,171.303,-108.853,169.148,45.315,158.538
C06478=1029.286,171.054,-108.831,169.145,45.317,158.538
C06479=1029.281,170.805,-108.808,169.141,45.320,158.538
C06480=1029.275,170.556,-108.785,169.139,45.322,158.538
C06481=1029.269,170.307,-108.762,169.136,45.325,158.538
C06482=1029.263,170.059,-108.740,169.132,45.327,158.538
C06483=1029.257,169.810,-108.717,169.128,45.329,158.538
C06484=1029.251,169.561,-108.694,169.126,45.332,158.539
C06485=1029.246,169.312,-108.671,169.123,45.334,158.539
C06486=1029.239,169.063,-108.648,169.119,45.337,158.539
C06487=1029.234,168.814,-108.626,169.117,45.339,158.539
C06488=1029.228,168.565,-108.603,169.113,45.342,158.539
C06489=1029.222,168.316,-108.580,169.110,45.344,158.540
C06490=1029.216,168.068,-108.558,169.108,45.346,158.540
C06491=1029.210,167.819,-108.535,169.104,45.349,158.540
C06492=1029.205,167.569,-108.513,169.101,45.351,158.540
C06493=1029.199,167.320,-108.490,169.097,45.354,158.540
C06494=1029.192,167.072,-108.467,169.095,45.356,158.540
C06495=1029.187,166.823,-108.444,169.091,45.359,158.541
C06496=1029.181,166.574,-108.421,169.088,45.361,158.541
C06497=1029.175,166.324,-108.399,169.086,45.363,158.541
C06498=1029.169,166.076,-108.377,169.082,45.366,158.541
C06499=1029.163,165.827,-108.354,169.079,45.368,158.541
C06500=1029.158,165.579,-108.331,169.076,45.371,158.541
C06501=1029.152,165.329,-108.310,169.073,45.373,158.541
C06502=1029.146,165.081,-108.287,169.070,45.375,158.542
C06503=1029.141,164.832,-108.264,169.067,45.378,158.542
C06504=1029.135,164.583,-108.241,169.064,45.381,158.542
C06505=1029.129,164.334,-108.219,169.061,45.383,158.542
C06506=1029.123,164.085,-108.196,169.058,45.385,158.542
C06507=1029.117,163.836,-108.173,169.054,45.388,158.543
C06508=1029.112,163.586,-108.151,169.052,45.390,158.543
C06509=1029.106,163.338,-108.129,169.048,45.392,158.543
C06510=1029.100,163.090,-108.106,169.046,45.394,158.543
C06511=1029.095,162.840,-108.084,169.043,45.397,158.543
C06512=1029.088,162.591,-108.062,169.039,45.400,158.543
C06513=1029.083,162.342,-108.039,169.037,45.402,158.544
C06514=1029.077,162.093,-108.016,169.033,45.404,158.544
C06515=1029.072,161.845,-107.994,169.031,45.407,158.544
C06516=1029.066,161.596,-107.972,169.027,45.409,158.544
C06517=1029.060,161.347,-107.949,169.024,45.412,158.544
C06518=1029.055,161.097,-107.927,169.022,45.414,158.544
C06519=1029.048,160.849,-107.905,169.018,45.416,158.544
C06520=1029.043,160.600,-107.882,169.016,45.419,158.545
C06521=1029.038,160.351,-107.860,169.012,45.421,158.545
C06522=1029.032,160.102,-107.837,169.009,45.424,158.545
C06523=1029.026,159.853,-107.815,169.006,45.426,158.545
C06524=1029.020,159.604,-107.792,169.003,45.429,158.545
C06525=1029.014,159.355,-107.771,169.001,45.431,158.546
C06526=1029.009,159.106,-107.748,168.997,45.434,158.546
C06527=1029.003,158.857,-107.727,168.994,45.437,158.546
C06528=1028.996,158.608,-107.705,168.991,45.439,158.546
C06529=1028.991,158.359,-107.682,168.988,45.442,158.546
C06530=1028.984,158.110,-107.660,168.985,45.445,158.547
C06531=1028.979,157.861,-107.639,168.982,45.447,158.547
C06532=1028.972,157.613,-107.617,168.979,45.449,158.547
C06533=1028.967,157.363,-107.594,168.977,45.452,158.547
C06534=1028.961,157.114,-107.573,168.973,45.454,158.547
C06535=1028.955,156.865,-107.551,168.970,45.457,158.548
C06536=1028.948,156.581,-107.526,168.967,45.460,158.548
C06537=1028.941,156.297,-107.501,168.963,45.463,158.548
C06538=1028.935,156.013,-107.476,168.960,45.466,158.548
C06539=1028.928,155.728,-107.451,168.957,45.469,158.549
C06540=1028.922,155.480,-107.429,168.954,45.472,158.549
C06541=1028.916,155.231,-107.408,168.951,45.474,158.549
C06542=1028.910,154.982,-107.385,168.948,45.477,158.549
C06543=1028.904,154.732,-107.363,168.944,45.479,158.549
C06544=1028.899,154.484,-107.342,168.942,45.482,158.550
C06545=1028.893,154.235,-107.320,168.939,45.484,158.550
C06546=1028.887,153.985,-107.298,168.936,45.487,158.550
C06547=1028.881,153.737,-107.276,168.933,45.490,158.550
C06548=1028.875,153.488,-107.254,168.931,45.492,158.550
C06549=1028.869,153.239,-107.233,168.927,45.495,158.551
C06550=1028.863,152.990,-107.211,168.924,45.498,158.551
C06551=1028.857,152.741,-107.189,168.922,45.500,158.551
C06552=1028.851,152.492,-107.168,168.918,45.503,158.551
C06553=1028.846,152.242,-107.146,168.916,45.505,158.551
C06554=1028.839,151.993,-107.124,168.913,45.508,158.552
C06555=1028.834,151.745,-107.103,168.909,45.511,158.552
C06556=1028.828,151.496,-107.081,168.907,45.513,158.552
C06557=1028.821,151.247,-107.059,168.904,45.516,158.552
C06558=1028.815,150.998,-107.037,168.901,45.519,158.553
C06559=1028.810,150.749,-107.016,168.898,45.522,158.553
C06560=1028.803,150.500,-106.994,168.895,45.524,158.553
C06561=1028.797,150.251,-106.973,168.892,45.526,158.553
C06562=1028.792,150.002,-106.951,168.889,45.529,158.553
C06563=1028.786,149.753,-106.929,168.887,45.532,158.554
C06564=1028.780,149.504,-106.908,168.883,45.534,158.554
C06565=1028.775,149.255,-106.886,168.881,45.537,158.554
C06566=1028.768,149.006,-106.865,168.878,45.540,158.554
C06567=1028.762,148.757,-106.843,168.875,45.542,158.555
C06568=1028.757,148.508,-106.822,168.872,45.545,158.555
C06569=1028.750,148.259,-106.800,168.869,45.547,158.555
C06570=1028.745,148.010,-106.780,168.866,45.550,158.555
C06571=1028.739,147.761,-106.758,168.863,45.553,158.555
C06572=1028.733,147.511,-106.736,168.861,45.556,158.556
C06573=1028.727,147.263,-106.715,168.857,45.558,158.556
C06574=1028.721,147.014,-106.694,168.855,45.561,158.556
C06575=1028.715,146.765,-106.672,168.852,45.564,158.556
C06576=1028.709,146.516,-106.651,168.849,45.566,158.556
C06577=1028.703,146.267,-106.629,168.846,45.569,158.557
C06578=1028.698,146.018,-106.608,168.843,45.571,158.557
C06579=1028.692,145.769,-106.587,168.840,45.574,158.557
C06580=1028.686,145.519,-106.565,168.838,45.577,158.557
C06581=1028.680,145.271,-106.544,168.835,45.580,158.558
C06582=1028.673,145.022,-106.523,168.831,45.583,158.558
C06583=1028.667,144.772,-106.502,168.829,45.585,158.558
C06584=1028.662,144.524,-106.481,168.826,45.588,158.558
C06585=1028.656,144.274,-106.459,168.823,45.590,158.558
C06586=1028.650,144.026,-106.438,168.820,45.593,158.559
C06587=1028.644,143.776,-106.417,168.818,45.596,158.559
C06588=1028.638,143.528,-106.396,168.814,45.599,158.559
C06589=1028.632,143.279,-106.375,168.812,45.601,158.559
C06590=1028.626,143.029,-106.354,168.809,45.604,158.560
C06591=1028.620,142.780,-106.332,168.807,45.607,158.560
C06592=1028.614,142.531,-106.311,168.803,45.609,158.560
C06593=1028.609,142.283,-106.289,168.801,45.612,158.560
C06594=1028.602,142.033,-106.269,168.798,45.615,158.561
C06595=1028.596,141.785,-106.248,168.795,45.617,158.561
C06596=1028.590,141.535,-106.226,168.792,45.620,158.561
C06597=1028.585,141.286,-106.206,168.790,45.623,158.561
C06598=1028.579,141.037,-106.184,168.786,45.626,158.562
C06599=1028.574,140.788,-106.163,168.784,45.628,158.562
C06600=1028.566,140.503,-106.139,168.781,45.632,158.562
C06601=1028.560,140.219,-106.115,168.778,45.634,158.562
C06602=1028.552,139.934,-106.091,168.774,45.637,158.563
C06603=1028.546,139.650,-106.067,168.771,45.640,158.563
C06604=1028.540,139.401,-106.046,168.768,45.643,158.563
C06605=1028.534,139.152,-106.025,168.766,45.646,158.563
C06606=1028.529,138.903,-106.004,168.762,45.649,158.563
C06607=1028.523,138.654,-105.982,168.760,45.651,158.564
C06608=1028.517,138.405,-105.962,168.757,45.654,158.564
C06609=1028.511,138.156,-105.941,168.754,45.657,158.564
C06610=1028.505,137.907,-105.921,168.751,45.660,158.565
C06611=1028.498,137.658,-105.899,168.749,45.663,158.565
C06612=1028.493,137.408,-105.879,168.745,45.665,158.565
C06613=1028.486,137.160,-105.858,168.743,45.668,158.565
C06614=1028.481,136.910,-105.837,168.740,45.671,158.565
C06615=1028.475,136.661,-105.815,168.738,45.673,158.566
C06616=1028.469,136.412,-105.795,168.734,45.676,158.566
C06617=1028.463,136.163,-105.774,168.732,45.679,158.566
C06618=1028.457,135.914,-105.753,168.729,45.682,158.566
C06619=1028.451,135.665,-105.733,168.727,45.684,158.567
C06620=1028.445,135.416,-105.712,168.723,45.687,158.567
C06621=1028.439,135.167,-105.691,168.721,45.690,158.567
C06622=1028.433,134.917,-105.671,168.718,45.693,158.567
C06623=1028.427,134.669,-105.650,168.715,45.696,158.568
C06624=1028.421,134.419,-105.629,168.712,45.699,158.568
C06625=1028.416,134.171,-105.608,168.710,45.701,158.568
C06626=1028.409,133.921,-105.588,168.707,45.704,158.568
C06627=1028.404,133.672,-105.567,168.704,45.707,158.569
C06628=1028.397,133.423,-105.546,168.701,45.710,158.569
C06629=1028.392,133.174,-105.525,168.699,45.712,158.569
C06630=1028.386,132.925,-105.505,168.696,45.714,158.569
C06631=1028.380,132.676,-105.484,168.693,45.717,158.570
C06632=1028.374,132.427,-105.464,168.691,45.720,158.570
C06633=1028.368,132.178,-105.443,168.688,45.723,158.570
C06634=1028.362,131.928,-105.422,168.685,45.726,158.570
C06635=1028.356,131.680,-105.402,168.682,45.729,158.571
C06636=1028.350,131.430,-105.381,168.680,45.731,158.571
C06637=1028.344,131.182,-105.361,168.676,45.734,158.571
C06638=1028.339,130.933,-105.340,168.674,45.737,158.571
C06639=1028.332,130.684,-105.319,168.672,45.740,158.572
C06640=1028.327,130.435,-105.299,168.669,45.743,158.572
C06641=1028.320,130.185,-105.278,168.666,45.745,158.572
C06642=1028.314,129.936,-105.258,168.663,45.748,158.572
C06643=1028.309,129.687,-105.238,168.661,45.751,158.573
C06644=1028.302,129.438,-105.217,168.658,45.754,158.573
C06645=1028.296,129.189,-105.198,168.655,45.756,158.573
C06646=1028.290,128.940,-105.176,168.652,45.759,158.573
C06647=1028.284,128.691,-105.157,168.650,45.762,158.574
C06648=1028.278,128.442,-105.136,168.647,45.766,158.574
C06649=1028.272,128.192,-105.116,168.645,45.768,158.574
C06650=1028.266,127.944,-105.096,168.641,45.771,158.574
C06651=1028.260,127.695,-105.076,168.639,45.774,158.575
C06652=1028.254,127.445,-105.055,168.636,45.777,158.575
C06653=1028.248,127.196,-105.035,168.634,45.780,158.575
C06654=1028.242,126.947,-105.015,168.630,45.783,158.575
C06655=1028.235,126.698,-104.995,168.628,45.785,158.576
C06656=1028.229,126.449,-104.975,168.625,45.788,158.576
C06657=1028.224,126.200,-104.954,168.622,45.791,158.576
C06658=1028.217,125.950,-104.934,168.619,45.794,158.576
C06659=1028.211,125.702,-104.914,168.617,45.797,158.577
C06660=1028.205,125.453,-104.894,168.615,45.800,158.577
C06661=1028.200,125.203,-104.873,168.612,45.803,158.577
C06662=1028.194,124.954,-104.853,168.609,45.805,158.578
C06663=1028.188,124.705,-104.833,168.606,45.808,158.578
C06664=1028.180,124.421,-104.810,168.603,45.811,158.578
C06665=1028.173,124.136,-104.787,168.600,45.815,158.579
C06666=1028.166,123.851,-104.764,168.597,45.818,158.579
C06667=1028.160,123.566,-104.741,168.595,45.821,158.579
C06668=1028.154,123.318,-104.721,168.591,45.824,158.579
C06669=1028.148,123.069,-104.701,168.589,45.827,158.580
C06670=1028.142,122.818,-104.681,168.586,45.830,158.580
C06671=1028.136,122.570,-104.661,168.584,45.833,158.580
C06672=1028.130,122.321,-104.641,168.580,45.835,158.580
C06673=1028.124,122.072,-104.621,168.578,45.838,158.581
C06674=1028.118,121.822,-104.600,168.576,45.841,158.581
C06675=1028.113,121.573,-104.580,168.573,45.844,158.581
C06676=1028.107,121.325,-104.560,168.570,45.847,158.581
C06677=1028.101,121.076,-104.540,168.567,45.849,158.582
C06678=1028.094,120.826,-104.520,168.565,45.852,158.582
C06679=1028.088,120.577,-104.500,168.562,45.855,158.582
C06680=1028.083,120.328,-104.480,168.559,45.858,158.582
C06681=1028.077,120.079,-104.460,168.557,45.860,158.583
C06682=1028.071,119.830,-104.440,168.554,45.863,158.583
C06683=1028.064,119.580,-104.419,168.551,45.866,158.583
C06684=1028.059,119.331,-104.400,168.549,45.869,158.583
C06685=1028.053,119.082,-104.380,168.546,45.872,158.584
C06686=1028.047,118.833,-104.360,168.544,45.874,158.584
C06687=1028.041,118.584,-104.340,168.540,45.877,158.584
C06688=1028.035,118.335,-104.319,168.538,45.881,158.585
C06689=1028.029,118.085,-104.300,168.536,45.884,158.585
C06690=1028.023,117.837,-104.280,168.533,45.886,158.585
C06691=1028.018,117.587,-104.260,168.531,45.889,158.585
C06692=1028.012,117.339,-104.240,168.528,45.892,158.586
C06693=1028.006,117.089,-104.220,168.525,45.895,158.586
C06694=1028.000,116.840,-104.200,168.523,45.898,158.586
C06695=1027.994,116.591,-104.180,168.521,45.900,158.586
C06696=1027.988,116.341,-104.161,168.517,45.903,158.587
C06697=1027.983,116.092,-104.140,168.515,45.906,158.587
C06698=1027.977,115.843,-104.120,168.512,45.909,158.587
C06699=1027.971,115.595,-104.100,168.510,45.912,158.587
C06700=1027.965,115.345,-104.081,168.507,45.914,158.588
C06701=1027.959,115.096,-104.061,168.504,45.917,158.588
C06702=1027.952,114.847,-104.041,168.502,45.919,158.588
C06703=1027.948,114.597,-104.021,168.499,45.922,158.588
C06704=1027.942,114.348,-104.001,168.496,45.925,158.589
C06705=1027.936,114.100,-103.981,168.494,45.928,158.589
C06706=1027.930,113.850,-103.962,168.492,45.930,158.589
C06707=1027.924,113.601,-103.942,168.488,45.933,158.589
C06708=1027.918,113.352,-103.922,168.486,45.936,158.590
C06709=1027.913,113.103,-103.902,168.484,45.939,158.590
C06710=1027.907,112.854,-103.882,168.482,45.941,158.590
C06711=1027.901,112.604,-103.863,168.478,45.944,158.590
C06712=1027.895,112.355,-103.843,168.476,45.947,158.591
C06713=1027.888,112.106,-103.824,168.473,45.951,158.591
C06714=1027.882,111.857,-103.804,168.471,45.953,158.591
C06715=1027.877,111.608,-103.785,168.469,45.956,158.592
C06716=1027.871,111.359,-103.765,168.465,45.959,158.592
C06717=1027.865,111.109,-103.746,168.463,45.962,158.592
C06718=1027.859,110.861,-103.726,168.461,45.964,158.592
C06719=1027.853,110.611,-103.706,168.458,45.967,158.593
C06720=1027.847,110.362,-103.686,168.455,45.970,158.593
C06721=1027.841,110.113,-103.667,168.452,45.973,158.593
C06722=1027.834,109.863,-103.648,168.450,45.976,158.593
C06723=1027.828,109.614,-103.628,168.448,45.979,158.594
C06724=1027.823,109.365,-103.609,168.445,45.982,158.594
C06725=1027.817,109.116,-103.589,168.442,45.985,158.594
C06726=1027.810,108.867,-103.570,168.439,45.988,158.594
C06727=1027.805,108.617,-103.551,168.437,45.991,158.595
C06728=1027.798,108.333,-103.528,168.434,45.994,158.595
C06729=1027.791,108.048,-103.506,168.431,45.998,158.595
C06730=1027.784,107.763,-103.485,168.428,46.001,158.596
C06731=1027.777,107.478,-103.463,168.426,46.004,158.596
C06732=1027.771,107.229,-103.443,168.422,46.007,158.596
C06733=1027.765,106.980,-103.424,168.420,46.010,158.597
C06734=1027.759,106.731,-103.405,168.418,46.013,158.597
C06735=1027.753,106.481,-103.385,168.415,46.016,158.597
C06736=1027.746,106.233,-103.366,168.413,46.019,158.597
C06737=1027.741,105.983,-103.347,168.409,46.022,158.598
C06738=1027.735,105.734,-103.328,168.407,46.025,158.598
C06739=1027.728,105.485,-103.308,168.405,46.027,158.598
C06740=1027.723,105.236,-103.289,168.402,46.030,158.598
C06741=1027.717,104.987,-103.270,168.399,46.033,158.599
C06742=1027.711,104.737,-103.250,168.397,46.036,158.599
C06743=1027.705,104.489,-103.231,168.394,46.039,158.599
C06744=1027.699,104.239,-103.212,168.392,46.042,158.600
C06745=1027.693,103.990,-103.193,168.390,46.045,158.600
C06746=1027.687,103.741,-103.174,168.386,46.048,158.600
C06747=1027.681,103.491,-103.155,168.384,46.050,158.600
C06748=1027.675,103.242,-103.135,168.382,46.053,158.601
C06749=1027.669,102.993,-103.116,168.379,46.056,158.601
C06750=1027.663,102.744,-103.097,168.377,46.060,158.601
C06751=1027.657,102.494,-103.078,168.374,46.062,158.602
C06752=1027.651,102.245,-103.059,168.371,46.065,158.602
C06753=1027.645,101.996,-103.039,168.369,46.068,158.602
C06754=1027.639,101.747,-103.020,168.367,46.071,158.602
C06755=1027.634,101.498,-103.001,168.363,46.074,158.603
C06756=1027.628,101.249,-102.982,168.361,46.076,158.603
C06757=1027.622,101.000,-102.963,168.359,46.079,158.603
C06758=1027.616,100.750,-102.944,168.356,46.082,158.603
C06759=1027.610,100.501,-102.925,168.353,46.085,158.604
C06760=1027.604,100.252,-102.906,168.351,46.088,158.604
C06761=1027.598,100.003,-102.886,168.348,46.091,158.604
C06762=1027.592,99.754,-102.867,168.346,46.094,158.605
C06763=1027.586,99.504,-102.848,168.344,46.097,158.605
C06764=1027.580,99.255,-102.829,168.340,46.100,158.605
C06765=1027.574,99.006,-102.810,168.338,46.102,158.605
C06766=1027.568,98.757,-102.792,168.336,46.106,158.606
C06767=1027.561,98.508,-102.773,168.333,46.109,158.606
C06768=1027.555,98.258,-102.754,168.331,46.111,158.606
C06769=1027.549,98.009,-102.735,168.328,46.114,158.606
C06770=1027.544,97.760,-102.717,168.325,46.118,158.607
C06771=1027.538,97.511,-102.698,168.323,46.120,158.607
C06772=1027.531,97.261,-102.680,168.320,46.123,158.607
C06773=1027.526,97.012,-102.660,168.318,46.126,158.608
C06774=1027.519,96.763,-102.642,168.315,46.129,158.608
C06775=1027.514,96.513,-102.622,168.313,46.133,158.608
C06776=1027.507,96.264,-102.604,168.310,46.135,158.608
C06777=1027.501,96.015,-102.584,168.308,46.138,158.609
C06778=1027.495,95.766,-102.566,168.305,46.141,158.609
C06779=1027.489,95.517,-102.547,168.303,46.144,158.609
C06780=1027.483,95.268,-102.528,168.301,46.147,158.610
C06781=1027.477,95.019,-102.510,168.297,46.150,158.610
C06782=1027.471,94.769,-102.492,168.295,46.153,158.610
C06783=1027.465,94.520,-102.472,168.293,46.156,158.610
C06784=1027.459,94.271,-102.454,168.290,46.159,158.611
C06785=1027.453,94.021,-102.435,168.287,46.161,158.611
C06786=1027.447,93.772,-102.416,168.285,46.165,158.611
C06787=1027.441,93.524,-102.398,168.282,46.168,158.612
C06788=1027.435,93.274,-102.378,168.280,46.170,158.612
C06789=1027.429,93.024,-102.360,168.278,46.173,158.612
C06790=1027.423,92.775,-102.341,168.274,46.176,158.612
C06791=1027.417,92.526,-102.323,168.272,46.179,158.613
C06792=1027.411,92.242,-102.301,168.269,46.183,158.613
C06793=1027.403,91.956,-102.280,168.267,46.186,158.613
C06794=1027.397,91.672,-102.259,168.264,46.189,158.614
C06795=1027.390,91.387,-102.237,168.261,46.193,158.614
C06796=1027.384,91.138,-102.218,168.259,46.195,158.614
C06797=1027.378,90.888,-102.200,168.255,46.198,158.614
C06798=1027.372,90.640,-102.182,168.253,46.201,158.615
C06799=1027.366,90.390,-102.163,168.251,46.204,158.615
C06800=1027.360,90.141,-102.144,168.249,46.206,158.615
C06801=1027.355,89.891,-102.125,168.246,46.210,158.616
C06802=1027.348,89.642,-102.107,168.244,46.213,158.616
C06803=1027.342,89.394,-102.089,168.241,46.216,158.616
C06804=1027.336,89.144,-102.071,168.238,46.219,158.616
C06805=1027.330,88.895,-102.052,168.236,46.222,158.617
C06806=1027.323,88.646,-102.033,168.234,46.225,158.617
C06807=1027.318,88.395,-102.015,168.231,46.228,158.617
C06808=1027.312,88.147,-101.996,168.228,46.230,158.617
C06809=1027.306,87.897,-101.979,168.225,46.234,158.618
C06810=1027.300,87.648,-101.960,168.223,46.237,158.618
C06811=1027.293,87.398,-101.942,168.221,46.240,158.618
C06812=1027.287,87.149,-101.923,168.218,46.243,158.619
C06813=1027.281,86.901,-101.905,168.216,46.246,158.619
C06814=1027.275,86.651,-101.887,168.214,46.249,158.619
C06815=1027.269,86.402,-101.868,168.210,46.252,158.619
C06816=1027.262,86.152,-101.851,168.208,46.254,158.620
C06817=1027.257,85.904,-101.832,168.206,46.258,158.620
C06818=1027.251,85.654,-101.814,168.203,46.261,158.620
C06819=1027.245,85.405,-101.795,168.201,46.264,158.621
C06820=1027.239,85.155,-101.777,168.198,46.266,158.621
C06821=1027.233,84.907,-101.759,168.195,46.270,158.621
C06822=1027.227,84.657,-101.741,168.193,46.273,158.622
C06823=1027.220,84.408,-101.722,168.191,46.276,158.622
C06824=1027.215,84.159,-101.705,168.188,46.279,158.622
C06825=1027.208,83.910,-101.686,168.186,46.282,158.622
C06826=1027.202,83.660,-101.668,168.183,46.285,158.623
C06827=1027.196,83.411,-101.649,168.180,46.288,158.623
C06828=1027.190,83.162,-101.632,168.178,46.290,158.623
C06829=1027.184,82.913,-101.613,168.176,46.293,158.623
C06830=1027.178,82.663,-101.595,168.174,46.297,158.624
C06831=1027.172,82.414,-101.577,168.171,46.300,158.624
C06832=1027.166,82.165,-101.559,168.168,46.302,158.624
C06833=1027.160,81.915,-101.540,168.166,46.305,158.625
C06834=1027.155,81.666,-101.522,168.163,46.308,158.625
C06835=1027.149,81.416,-101.504,168.161,46.312,158.625
C06836=1027.142,81.167,-101.486,168.159,46.314,158.626
C06837=1027.137,80.918,-101.468,168.155,46.317,158.626
C06838=1027.130,80.669,-101.449,168.153,46.320,158.626
C06839=1027.124,80.419,-101.432,168.151,46.323,158.626
C06840=1027.119,80.170,-101.414,168.148,46.326,158.626
C06841=1027.112,79.921,-101.395,168.146,46.329,158.627
C06842=1027.106,79.671,-101.377,168.144,46.332,158.627
C06843=1027.100,79.423,-101.359,168.141,46.335,158.627
C06844=1027.094,79.173,-101.341,168.138,46.338,158.628
C06845=1027.088,78.924,-101.323,168.136,46.340,158.628
C06846=1027.082,78.675,-101.305,168.134,46.343,158.628
C06847=1027.076,78.425,-101.287,168.130,46.346,158.628
C06848=1027.070,78.176,-101.269,168.128,46.350,158.629
C06849=1027.064,77.927,-101.251,168.126,46.352,158.629
C06850=1027.058,77.677,-101.233,168.124,46.355,158.629
C06851=1027.052,77.428,-101.215,168.121,46.358,158.630
C06852=1027.046,77.179,-101.197,168.118,46.361,158.630
C06853=1027.040,76.930,-101.179,168.116,46.364,158.630
C06854=1027.034,76.681,-101.161,168.113,46.367,158.630
C06855=1027.028,76.431,-101.143,168.111,46.370,158.631
C06856=1027.022,76.146,-101.123,168.108,46.374,158.631
C06857=1027.014,75.861,-101.102,168.105,46.377,158.631
C06858=1027.008,75.576,-101.082,168.103,46.380,158.632
C06859=1027.001,75.292,-101.062,168.100,46.384,158.632
C06860=1026.994,75.042,-101.044,168.097,46.387,158.632
C06861=1026.989,74.793,-101.027,168.095,46.390,158.633
C06862=1026.982,74.544,-101.009,168.092,46.393,158.633
C06863=1026.976,74.294,-100.991,168.090,46.396,158.633
C06864=1026.970,74.046,-100.973,168.087,46.399,158.633
C06865=1026.964,73.796,-100.955,168.085,46.402,158.634
C06866=1026.958,73.547,-100.938,168.083,46.405,158.634
C06867=1026.952,73.297,-100.920,168.080,46.408,158.634
C06868=1026.946,73.047,-100.902,168.077,46.411,158.635
C06869=1026.940,72.799,-100.885,168.075,46.413,158.635
C06870=1026.933,72.549,-100.867,168.072,46.417,158.635
C06871=1026.928,72.300,-100.849,168.070,46.420,158.635
C06872=1026.922,72.050,-100.831,168.068,46.423,158.636
C06873=1026.915,71.802,-100.814,168.064,46.426,158.636
C06874=1026.909,71.552,-100.796,168.062,46.429,158.636
C06875=1026.904,71.303,-100.778,168.060,46.432,158.637
C06876=1026.898,71.054,-100.760,168.057,46.435,158.637
C06877=1026.891,70.805,-100.743,168.055,46.438,158.637
C06878=1026.885,70.555,-100.725,168.053,46.440,158.637
C06879=1026.880,70.306,-100.708,168.050,46.444,158.638
C06880=1026.874,70.056,-100.690,168.047,46.447,158.638
C06881=1026.867,69.808,-100.673,168.045,46.450,158.638
C06882=1026.861,69.558,-100.655,168.043,46.452,158.638
C06883=1026.856,69.309,-100.637,168.040,46.455,158.639
C06884=1026.849,69.059,-100.620,168.038,46.459,158.639
C06885=1026.843,68.810,-100.603,168.036,46.462,158.639
C06886=1026.837,68.561,-100.585,168.032,46.465,158.640
C06887=1026.831,68.312,-100.568,168.030,46.467,158.640
C06888=1026.825,68.062,-100.550,168.028,46.471,158.640
C06889=1026.820,67.812,-100.533,168.025,46.474,158.640
C06890=1026.813,67.563,-100.516,168.023,46.477,158.641
C06891=1026.807,67.314,-100.498,168.020,46.479,158.641
C06892=1026.800,67.065,-100.481,168.017,46.483,158.641
C06893=1026.795,66.815,-100.463,168.015,46.486,158.642
C06894=1026.789,66.566,-100.445,168.013,46.489,158.642
C06895=1026.782,66.317,-100.428,168.010,46.492,158.642
C06896=1026.776,66.067,-100.410,168.008,46.495,158.642
C06897=1026.770,65.818,-100.394,168.006,46.498,158.643
C06898=1026.764,65.568,-100.376,168.002,46.501,158.643
C06899=1026.758,65.319,-100.359,168.000,46.504,158.643
C06900=1026.752,65.070,-100.341,167.998,46.507,158.644
C06901=1026.746,64.821,-100.324,167.995,46.510,158.644
C06902=1026.739,64.571,-100.306,167.993,46.513,158.644
C06903=1026.733,64.322,-100.290,167.991,46.516,158.644
C06904=1026.728,64.073,-100.272,167.988,46.519,158.645
C06905=1026.721,63.823,-100.255,167.985,46.522,158.645
C06906=1026.716,63.574,-100.237,167.983,46.525,158.645
C06907=1026.709,63.325,-100.220,167.981,46.528,158.645
C06908=1026.704,63.075,-100.203,167.978,46.531,158.646
C06909=1026.697,62.826,-100.186,167.976,46.534,158.646
C06910=1026.690,62.577,-100.169,167.972,46.537,158.646
C06911=1026.685,62.327,-100.152,167.971,46.541,158.647
C06912=1026.678,62.078,-100.135,167.968,46.543,158.647
C06913=1026.672,61.829,-100.119,167.965,46.547,158.647
C06914=1026.666,61.579,-100.101,167.963,46.550,158.648
C06915=1026.660,61.330,-100.084,167.960,46.553,158.648
C06916=1026.653,61.080,-100.067,167.958,46.556,158.648
C06917=1026.647,60.831,-100.050,167.956,46.559,158.648
C06918=1026.640,60.582,-100.033,167.953,46.563,158.649
C06919=1026.634,60.333,-100.016,167.951,46.565,158.649
C06920=1026.628,60.047,-99.997,167.948,46.569,158.649
C06921=1026.621,59.763,-99.977,167.945,46.573,158.650
C06922=1026.613,59.478,-99.958,167.941,46.576,158.650
C06923=1026.607,59.192,-99.938,167.938,46.580,158.650
C06924=1026.600,58.944,-99.921,167.937,46.583,158.651
C06925=1026.594,58.694,-99.905,167.934,46.586,158.651
C06926=1026.587,58.445,-99.888,167.931,46.589,158.651
C06927=1026.582,58.195,-99.871,167.929,46.592,158.652
C06928=1026.575,57.946,-99.853,167.927,46.595,158.652
C06929=1026.569,57.696,-99.837,167.924,46.598,158.652
C06930=1026.563,57.448,-99.820,167.922,46.602,158.652
C06931=1026.557,57.198,-99.804,167.920,46.604,158.653
C06932=1026.551,56.949,-99.786,167.916,46.607,158.653
C06933=1026.545,56.699,-99.769,167.914,46.611,158.653
C06934=1026.538,56.450,-99.752,167.911,46.614,158.653
C06935=1026.532,56.200,-99.736,167.909,46.617,158.654
C06936=1026.526,55.951,-99.719,167.907,46.619,158.654
C06937=1026.520,55.701,-99.702,167.904,46.623,158.654
C06938=1026.514,55.453,-99.685,167.901,46.626,158.655
C06939=1026.507,55.203,-99.668,167.899,46.629,158.655
C06940=1026.501,54.954,-99.651,167.896,46.632,158.655
C06941=1026.496,54.704,-99.635,167.894,46.635,158.655
C06942=1026.490,54.455,-99.618,167.892,46.638,158.656
C06943=1026.483,54.205,-99.601,167.889,46.641,158.656
C06944=1026.477,53.956,-99.585,167.887,46.644,158.656
C06945=1026.471,53.707,-99.568,167.885,46.647,158.657
C06946=1026.465,53.457,-99.551,167.881,46.650,158.657
C06947=1026.459,53.208,-99.534,167.879,46.653,158.657
C06948=1026.453,52.959,-99.517,167.877,46.656,158.657
C06949=1026.446,52.709,-99.501,167.874,46.660,158.658
C06950=1026.440,52.460,-99.484,167.872,46.662,158.658
C06951=1026.435,52.210,-99.467,167.869,46.665,158.658
C06952=1026.429,51.962,-99.450,167.867,46.669,158.659
C06953=1026.422,51.712,-99.433,167.864,46.672,158.659
C06954=1026.416,51.462,-99.417,167.862,46.674,158.659
C06955=1026.410,51.214,-99.400,167.859,46.677,158.659
C06956=1026.405,50.964,-99.383,167.857,46.681,158.660
C06957=1026.398,50.714,-99.367,167.855,46.684,158.660
C06958=1026.392,50.465,-99.350,167.851,46.687,158.660
C06959=1026.386,50.216,-99.333,167.849,46.689,158.660
C06960=1026.380,49.966,-99.317,167.847,46.692,158.661
C06961=1026.374,49.717,-99.300,167.844,46.696,158.661
C06962=1026.368,49.467,-99.283,167.842,46.699,158.661
C06963=1026.362,49.218,-99.267,167.840,46.702,158.662
C06964=1026.356,48.969,-99.250,167.836,46.705,158.662
C06965=1026.350,48.720,-99.233,167.834,46.707,158.662
C06966=1026.344,48.470,-99.216,167.832,46.711,158.662
C06967=1026.338,48.220,-99.200,167.829,46.714,158.663
C06968=1026.332,47.972,-99.183,167.827,46.717,158.663
C06969=1026.326,47.722,-99.167,167.825,46.719,158.663
C06970=1026.320,47.473,-99.150,167.821,46.722,158.663
C06971=1026.314,47.224,-99.133,167.819,46.725,158.664
C06972=1026.308,46.974,-99.116,167.817,46.729,158.664
C06973=1026.302,46.724,-99.100,167.815,46.732,158.664
C06974=1026.296,46.475,-99.084,167.812,46.735,158.664
C06975=1026.290,46.226,-99.067,167.810,46.737,158.665
C06976=1026.284,45.977,-99.051,167.807,46.740,158.665
C06977=1026.278,45.727,-99.034,167.804,46.743,158.665
C06978=1026.272,45.477,-99.017,167.802,46.746,158.665
C06979=1026.266,45.228,-99.001,167.800,46.749,158.666
C06980=1026.260,44.979,-98.985,167.797,46.753,158.666
C06981=1026.254,44.730,-98.968,167.795,46.755,158.666
C06982=1026.248,44.480,-98.951,167.792,46.758,158.666
C06983=1026.243,44.231,-98.934,167.789,46.761,158.667
C06984=1026.235,43.946,-98.915,167.787,46.764,158.667
C06985=1026.229,43.660,-98.897,167.784,46.768,158.667
C06986=1026.222,43.375,-98.878,167.781,46.771,158.668
C06987=1026.216,43.090,-98.859,167.778,46.774,158.668
C06988=1026.209,42.840,-98.843,167.776,46.777,158.668
C06989=1026.203,42.591,-98.826,167.773,46.780,158.668
C06990=1026.197,42.341,-98.809,167.770,46.784,158.669
C06991=1026.191,42.092,-98.793,167.768,46.787,158.669
C06992=1026.185,41.843,-98.777,167.766,46.789,158.669
C06993=1026.179,41.593,-98.761,167.763,46.792,158.669
C06994=1026.173,41.344,-98.744,167.761,46.796,158.670
C06995=1026.166,41.095,-98.729,167.759,46.799,158.670
C06996=1026.160,40.845,-98.712,167.755,46.802,158.670
C06997=1026.154,40.596,-98.696,167.753,46.804,158.670
C06998=1026.148,40.346,-98.680,167.751,46.808,158.671
C06999=1026.142,40.096,-98.664,167.748,46.811,158.671
C07000=1026.136,39.847,-98.648,167.746,46.814,158.671
C07001=1026.130,39.598,-98.632,167.743,46.817,158.671
C07002=1026.124,39.348,-98.615,167.740,46.820,158.672
C07003=1026.118,39.099,-98.599,167.739,46.823,158.672
C07004=1026.112,38.850,-98.583,167.735,46.826,158.672
C07005=1026.106,38.601,-98.567,167.733,46.829,158.673
C07006=1026.100,38.351,-98.551,167.731,46.832,158.673
C07007=1026.094,38.102,-98.535,167.728,46.835,158.673
C07008=1026.088,37.853,-98.518,167.726,46.838,158.673
C07009=1026.082,37.603,-98.502,167.724,46.841,158.674
C07010=1026.076,37.354,-98.486,167.720,46.844,158.674
C07011=1026.069,37.104,-98.469,167.718,46.847,158.674
C07012=1026.063,36.854,-98.454,167.716,46.850,158.674
C07013=1026.057,36.605,-98.438,167.713,46.854,158.675
C07014=1026.051,36.355,-98.422,167.711,46.856,158.675
C07015=1026.044,36.106,-98.406,167.708,46.859,158.675
C07016=1026.039,35.857,-98.390,167.706,46.863,158.676
C07017=1026.033,35.607,-98.374,167.703,46.866,158.676
C07018=1026.026,35.358,-98.359,167.700,46.869,158.676
C07019=1026.020,35.109,-98.342,167.698,46.872,158.676
C07020=1026.014,34.859,-98.326,167.695,46.875,158.677
C07021=1026.008,34.610,-98.311,167.693,46.878,158.677
C07022=1026.002,34.360,-98.295,167.691,46.881,158.677
C07023=1025.996,34.111,-98.279,167.688,46.885,158.677
C07024=1025.990,33.861,-98.264,167.685,46.887,158.678
C07025=1025.984,33.612,-98.248,167.682,46.890,158.678
C07026=1025.978,33.363,-98.231,167.680,46.893,158.678
C07027=1025.971,33.114,-98.216,167.678,46.897,158.679
C07028=1025.965,32.864,-98.200,167.675,46.900,158.679
C07029=1025.959,32.615,-98.184,167.673,46.903,158.679
C07030=1025.953,32.365,-98.168,167.669,46.906,158.679
C07031=1025.947,32.115,-98.153,167.668,46.909,158.680
C07032=1025.940,31.866,-98.137,167.665,46.912,158.680
C07033=1025.934,31.617,-98.121,167.662,46.915,158.680
C07034=1025.929,31.367,-98.105,167.660,46.918,158.680
C07035=1025.922,31.118,-98.089,167.657,46.922,158.681
C07036=1025.916,30.869,-98.073,167.655,46.924,158.681
C07037=1025.911,30.619,-98.058,167.653,46.927,158.681
C07038=1025.904,30.370,-98.042,167.649,46.930,158.681
C07039=1025.898,30.120,-98.026,167.647,46.934,158.682
C07040=1025.891,29.871,-98.011,167.645,46.937,158.682
C07041=1025.886,29.622,-97.995,167.642,46.940,158.682
C07042=1025.880,29.372,-97.979,167.640,46.942,158.682
C07043=1025.874,29.123,-97.964,167.637,46.945,158.683
C07044=1025.868,28.873,-97.948,167.635,46.949,158.683
C07045=1025.862,28.624,-97.932,167.632,46.952,158.683
C07046=1025.856,28.375,-97.916,167.629,46.955,158.683
C07047=1025.850,28.125,-97.901,167.627,46.958,158.684
C07048=1025.842,27.839,-97.883,167.624,46.961,158.684
C07049=1025.836,27.554,-97.865,167.621,46.964,158.684
C07050=1025.829,27.269,-97.847,167.618,46.968,158.684
C07051=1025.822,26.984,-97.829,167.615,46.972,158.685
C07052=1025.815,26.734,-97.814,167.613,46.975,158.685
C07053=1025.809,26.485,-97.798,167.610,46.979,158.685
C07054=1025.803,26.235,-97.783,167.608,46.981,158.686
C07055=1025.797,25.985,-97.767,167.605,46.984,158.686
C07056=1025.791,25.736,-97.752,167.602,46.987,158.686
C07057=1025.786,25.487,-97.737,167.600,46.991,158.686
C07058=1025.779,25.238,-97.721,167.597,46.994,158.687
C07059=1025.773,24.988,-97.706,167.595,46.997,158.687
C07060=1025.767,24.738,-97.690,167.592,47.000,158.687
C07061=1025.760,24.489,-97.675,167.590,47.003,158.687
C07062=1025.754,24.239,-97.660,167.588,47.006,158.688
C07063=1025.748,23.990,-97.644,167.584,47.009,158.688
C07064=1025.742,23.740,-97.629,167.582,47.013,158.688
C07065=1025.737,23.491,-97.614,167.579,47.016,158.688
C07066=1025.730,23.242,-97.598,167.577,47.018,158.689
C07067=1025.723,22.992,-97.583,167.574,47.022,158.689
C07068=1025.718,22.743,-97.567,167.572,47.025,158.689
C07069=1025.711,22.493,-97.552,167.570,47.028,158.690
C07070=1025.705,22.244,-97.536,167.566,47.031,158.690
C07071=1025.700,21.995,-97.522,167.564,47.034,158.690
C07072=1025.693,21.746,-97.506,167.561,47.037,158.690
C07073=1025.687,21.496,-97.490,167.559,47.040,158.691
C07074=1025.681,21.246,-97.475,167.556,47.043,158.691
C07075=1025.675,20.996,-97.460,167.554,47.046,158.691
C07076=1025.669,20.748,-97.445,167.552,47.049,158.691
C07077=1025.663,20.498,-97.430,167.549,47.053,158.692
C07078=1025.657,20.248,-97.414,167.546,47.056,158.692
C07079=1025.651,19.999,-97.398,167.543,47.059,158.692
C07080=1025.644,19.749,-97.384,167.541,47.062,158.692
C07081=1025.639,19.500,-97.368,167.538,47.065,158.692
C07082=1025.633,19.250,-97.353,167.536,47.068,158.693
C07083=1025.626,19.001,-97.338,167.534,47.071,158.693
C07084=1025.620,18.752,-97.323,167.530,47.074,158.693
C07085=1025.614,18.502,-97.307,167.528,47.077,158.694
C07086=1025.608,18.253,-97.293,167.525,47.081,158.694
C07087=1025.602,18.003,-97.278,167.523,47.083,158.694
C07088=1025.595,17.753,-97.263,167.520,47.086,158.694
C07089=1025.590,17.503,-97.247,167.518,47.089,158.695
C07090=1025.584,17.255,-97.232,167.515,47.093,158.695
C07091=1025.577,17.005,-97.217,167.513,47.096,158.695
C07092=1025.571,16.756,-97.202,167.509,47.099,158.695
C07093=1025.565,16.506,-97.187,167.507,47.102,158.696
C07094=1025.560,16.257,-97.172,167.505,47.105,158.696
C07095=1025.553,16.007,-97.157,167.502,47.108,158.696
C07096=1025.547,15.758,-97.142,167.500,47.111,158.696
C07097=1025.540,15.508,-97.127,167.497,47.114,158.696
C07098=1025.535,15.259,-97.112,167.495,47.118,158.697
C07099=1025.529,15.009,-97.097,167.492,47.121,158.697
C07100=1025.523,14.759,-97.082,167.489,47.124,158.697
C07101=1025.516,14.511,-97.067,167.486,47.127,158.697
C07102=1025.510,14.261,-97.052,167.484,47.130,158.698
C07103=1025.504,14.011,-97.036,167.482,47.133,158.698
C07104=1025.498,13.762,-97.021,167.479,47.136,158.698
C07105=1025.492,13.513,-97.007,167.477,47.139,158.699
C07106=1025.486,13.263,-96.992,167.473,47.142,158.699
C07107=1025.480,13.013,-96.978,167.472,47.146,158.699
C07108=1025.474,12.764,-96.963,167.468,47.149,158.699
C07109=1025.468,12.514,-96.948,167.466,47.152,158.700
C07110=1025.461,12.265,-96.933,167.463,47.155,158.700
C07111=1025.456,12.016,-96.918,167.460,47.158,158.700
C07112=1025.448,11.731,-96.902,167.457,47.162,158.700
C07113=1025.441,11.448,-96.885,167.454,47.166,158.701
C07114=1025.434,11.163,-96.868,167.451,47.170,158.701
C07115=1025.427,10.880,-96.852,167.448,47.173,158.701
C07116=1025.420,10.630,-96.837,167.446,47.176,158.702
C07117=1025.414,10.381,-96.822,167.443,47.179,158.702
C07118=1025.408,10.132,-96.807,167.441,47.182,158.702
C07119=1025.402,9.881,-96.793,167.438,47.186,158.702
C07120=1025.396,9.632,-96.778,167.436,47.189,158.703
C07121=1025.390,9.383,-96.764,167.432,47.192,158.703
C07122=1025.384,9.133,-96.749,167.430,47.196,158.703
C07123=1025.378,8.884,-96.734,167.427,47.199,158.703
C07124=1025.371,8.635,-96.719,167.425,47.201,158.704
C07125=1025.365,8.385,-96.705,167.422,47.205,158.704
C07126=1025.359,8.136,-96.691,167.420,47.208,158.704
C07127=1025.352,7.886,-96.676,167.417,47.211,158.704
C07128=1025.347,7.637,-96.661,167.415,47.214,158.705
C07129=1025.341,7.387,-96.647,167.412,47.218,158.705
C07130=1025.334,7.137,-96.632,167.409,47.221,158.705
C07131=1025.328,6.888,-96.618,167.406,47.224,158.705
C07132=1025.322,6.638,-96.603,167.404,47.227,158.706
C07133=1025.317,6.389,-96.589,167.401,47.230,158.706
C07134=1025.310,6.139,-96.574,167.399,47.233,158.706
C07135=1025.304,5.890,-96.559,167.396,47.236,158.706
C07136=1025.298,5.641,-96.544,167.394,47.239,158.707
C07137=1025.292,5.390,-96.530,167.391,47.243,158.707
C07138=1025.285,5.142,-96.516,167.388,47.246,158.707
C07139=1025.279,4.892,-96.501,167.385,47.249,158.707
C07140=1025.274,4.642,-96.487,167.383,47.252,158.708
C07141=1025.267,4.393,-96.472,167.380,47.255,158.708
C07142=1025.261,4.144,-96.458,167.378,47.258,158.708
C07143=1025.255,3.894,-96.443,167.375,47.261,158.708
C07144=1025.250,3.645,-96.429,167.372,47.264,158.708
C07145=1025.243,3.395,-96.414,167.369,47.267,158.709
C07146=1025.237,3.145,-96.400,167.367,47.271,158.709
C07147=1025.231,2.896,-96.385,167.364,47.274,158.709
C07148=1025.224,2.646,-96.371,167.362,47.277,158.709
C07149=1025.219,2.397,-96.357,167.359,47.280,158.710
C07150=1025.212,2.147,-96.342,167.357,47.283,158.710
C07151=1025.207,1.898,-96.328,167.353,47.286,158.710
C07152=1025.200,1.648,-96.313,167.351,47.289,158.710
C07153=1025.195,1.399,-96.299,167.348,47.292,158.711
C07154=1025.189,1.149,-96.284,167.346,47.295,158.711
C07155=1025.183,0.900,-96.270,167.343,47.298,158.711
C07156=1025.177,0.650,-96.256,167.341,47.301,158.711
C07157=1025.171,0.400,-96.241,167.337,47.304,158.711
C07158=1025.165,0.151,-96.228,167.336,47.308,158.712
C07159=1025.158,-0.098,-96.213,167.332,47.311,158.712
C07160=1025.153,-0.347,-96.198,167.330,47.314,158.712
C07161=1025.146,-0.598,-96.184,167.327,47.317,158.712
C07162=1025.141,-0.847,-96.169,167.325,47.320,158.713
C07163=1025.135,-1.097,-96.155,167.322,47.323,158.713
C07164=1025.129,-1.346,-96.141,167.319,47.326,158.713
C07165=1025.123,-1.595,-96.127,167.316,47.329,158.713
C07166=1025.117,-1.845,-96.112,167.314,47.332,158.714
C07167=1025.111,-2.094,-96.098,167.311,47.335,158.714
C07168=1025.104,-2.344,-96.084,167.309,47.338,158.714
C07169=1025.099,-2.594,-96.070,167.306,47.341,158.714
C07170=1025.093,-2.843,-96.055,167.304,47.344,158.714
C07171=1025.087,-3.093,-96.041,167.300,47.347,158.715
C07172=1025.081,-3.342,-96.026,167.298,47.350,158.715
C07173=1025.075,-3.592,-96.012,167.295,47.353,158.715
C07174=1025.070,-3.842,-95.998,167.293,47.356,158.715
C07175=1025.063,-4.091,-95.984,167.290,47.360,158.716
C07176=1025.056,-4.368,-95.968,167.287,47.363,158.716
C07177=1025.050,-4.646,-95.953,167.284,47.367,158.716
C07178=1025.043,-4.923,-95.937,167.281,47.371,158.716
C07179=1025.036,-5.200,-95.923,167.278,47.374,158.716
C07180=1025.029,-5.454,-95.908,167.276,47.377,158.717
C07181=1025.024,-5.709,-95.893,167.272,47.380,158.717
C07182=1025.017,-5.963,-95.879,167.269,47.384,158.717
